LIN {X 0,Y 527.544,Z 904.757,A -85,B 0,C 180,E1 14975.921,E2 14975.921} C_VEL
LIN {X 0,Y 511.75,Z 974.005,A -85,B 0,C 180,E1 14979.243,E2 14979.243} C_VEL
LIN {X 0,Y 491.404,Z 1041.559,A -85,B 0,C 180,E1 14984.465,E2 14984.465} C_VEL
LIN {X 0,Y 471.066,Z 1101.33,A -85,B 0,C 180,E1 14991.676,E2 14991.676} C_VEL
LIN {X 0,Y 455.075,Z 1150.051,A -85,B 0,C 180,E1 15000.694,E2 15000.694} C_VEL
LIN {X 0,Y 446.451,Z 1183.071,A -85,B 0,C 180,E1 15010.14,E2 15010.14} C_VEL
LIN {X 0,Y 443.515,Z 1201.898,A -85,B 0,C 180,E1 15019.158,E2 15019.158} C_VEL
LIN {X 0,Y 443.252,Z 1209.224,A -85,B 0,C 180,E1 15027.056,E2 15027.056} C_VEL
LIN {X 0,Y 443.097,Z 1207.14,A -85,B 0,C 180,E1 15036.179,E2 15036.179} C_VEL
LIN {X 0,Y 443.595,Z 1202.243,A -85,B 0,C 180,E1 15040.591,E2 15040.591} C_VEL
LIN {X 0,Y 436.619,Z 1195.01,A -85,B 0,C 180,E1 15045.026,E2 15045.026} C_VEL
LIN {X 0,Y 442.886,Z 1167.282,A -85,B 0,C 180,E1 15055.338,E2 15055.338} C_VEL
LIN {X 0,Y 455.534,Z 1125.939,A -85,B 0,C 180,E1 15064.753,E2 15064.753} C_VEL
LIN {X 0,Y 473.85,Z 1072.374,A -85,B 0,C 180,E1 15072.653,E2 15072.653} C_VEL
LIN {X 0,Y 493.837,Z 1008.731,A -85,B 0,C 180,E1 15078.789,E2 15078.789} C_VEL
LIN {X 0,Y 512.572,Z 935.581,A -85,B 0,C 180,E1 15083.187,E2 15083.187} C_VEL
LIN {X 0,Y 518.028,Z 903.153,A -85,B 0,C 180,E1 15084.629,E2 15084.629} C_VEL
LIN {X 0,Y 493.673,Z 851.518,A -85,B 0,C 180,E1 15091.51,E2 15091.51} C_VEL
LIN {X 0,Y 466.915,Z 810.429,A -85,B 0,C 180,E1 15099.517,E2 15099.517} C_VEL
LIN {X 0,Y 448.656,Z 787.138,A -85,B 0,C 180,E1 15107.046,E2 15107.046} C_VEL
LIN {X 0,Y 439.151,Z 774.402,A -85,B 0,C 180,E1 15113.435,E2 15113.435} C_VEL
LIN {X 0,Y 434.536,Z 767.06,A -85,B 0,C 180,E1 15121.02,E2 15121.02} C_VEL
LIN {X 0,Y 434.845,Z 769.422,A -85,B 0,C 180,E1 15127.285,E2 15127.285} C_VEL
LIN {X 0,Y 441.325,Z 777.842,A -85,B 0,C 180,E1 15134.513,E2 15134.513} C_VEL
LIN {X 0,Y 452.767,Z 792.076,A -85,B 0,C 180,E1 15141.061,E2 15141.061} C_VEL
LIN {X 0,Y 474.863,Z 822.437,A -85,B 0,C 180,E1 15149.239,E2 15149.239} C_VEL
LIN {X 0,Y 501.419,Z 867.679,A -85,B 0,C 180,E1 15156.98,E2 15156.98} C_VEL
LIN {X 0,Y 517.133,Z 907.005,A -85,B 0,C 180,E1 15161.858,E2 15161.858} C_VEL
LIN {X 0,Y 499.871,Z 981.761,A -85,B 0,C 180,E1 15165.794,E2 15165.794} C_VEL
LIN {X 0,Y 479.961,Z 1047.78,A -85,B 0,C 180,E1 15171.441,E2 15171.441} C_VEL
LIN {X 0,Y 460.575,Z 1103.811,A -85,B 0,C 180,E1 15178.811,E2 15178.811} C_VEL
LIN {X 0,Y 446.089,Z 1147.116,A -85,B 0,C 180,E1 15187.518,E2 15187.518} C_VEL
LIN {X 0,Y 438.118,Z 1178.477,A -85,B 0,C 180,E1 15197.509,E2 15197.509} C_VEL
LIN {X 0,Y 435.402,Z 1195.059,A -85,B 0,C 180,E1 15207.008,E2 15207.008} C_VEL
LIN {X 0,Y 434.743,Z 1200.24,A -85,B 0,C 180,E1 15215.88,E2 15215.88} C_VEL
LIN {X 0,Y 435.395,Z 1194.776,A -85,B 0,C 180,E1 15225.145,E2 15225.145} C_VEL
LIN {X 0,Y 437.899,Z 1178.172,A -85,B 0,C 180,E1 15234.558,E2 15234.558} C_VEL
LIN {X 0,Y 446.288,Z 1146.664,A -85,B 0,C 180,E1 15244.563,E2 15244.563} C_VEL
LIN {X 0,Y 462.337,Z 1100.95,A -85,B 0,C 180,E1 15253.74,E2 15253.74} C_VEL
LIN {X 0,Y 483.029,Z 1043.534,A -85,B 0,C 180,E1 15261.229,E2 15261.229} C_VEL
LIN {X 0,Y 504.194,Z 977.942,A -85,B 0,C 180,E1 15266.717,E2 15266.717} C_VEL
LIN {X 0,Y 521.526,Z 904.091,A -85,B 0,C 180,E1 15270.64,E2 15270.64} C_VEL
LIN {X 0,Y 503.397,Z 862.252,A -85,B 0,C 180,E1 15277.068,E2 15277.068} C_VEL
LIN {X 0,Y 482.023,Z 826.723,A -85,B 0,C 180,E1 15285.517,E2 15285.517} C_VEL
LIN {X 0,Y 470.998,Z 812.054,A -85,B 0,C 180,E1 15291.649,E2 15291.649} C_VEL
LIN {X 0,Y 464.92,Z 803.945,A -85,B 0,C 180,E1 15297.527,E2 15297.527} C_VEL
LIN {X 0,Y 463.82,Z 803.136,A -85,B 0,C 180,E1 15306.379,E2 15306.379} C_VEL
LIN {X 0,Y 468.95,Z 809.648,A -85,B 0,C 180,E1 15312.592,E2 15312.592} C_VEL
LIN {X 0,Y 482.636,Z 828.099,A -85,B 0,C 180,E1 15320.554,E2 15320.554} C_VEL
LIN {X 0,Y 504.042,Z 862.875,A -85,B 0,C 180,E1 15328.764,E2 15328.764} C_VEL
LIN {X 0,Y 522.75,Z 905.365,A -85,B 0,C 180,E1 15335.174,E2 15335.174} C_VEL
LIN {X 0,Y 505.795,Z 977.464,A -85,B 0,C 180,E1 15338.719,E2 15338.719} C_VEL
LIN {X 0,Y 484.736,Z 1044.49,A -85,B 0,C 180,E1 15344.039,E2 15344.039} C_VEL
LIN {X 0,Y 463.733,Z 1103.615,A -85,B 0,C 180,E1 15351.37,E2 15351.37} C_VEL
LIN {X 0,Y 447.299,Z 1151.661,A -85,B 0,C 180,E1 15360.552,E2 15360.552} C_VEL
LIN {X 0,Y 438.391,Z 1184.327,A -85,B 0,C 180,E1 15370.287,E2 15370.287} C_VEL
LIN {X 0,Y 435.524,Z 1203.155,A -85,B 0,C 180,E1 15379.971,E2 15379.971} C_VEL
LIN {X 0,Y 434.854,Z 1209.594,A -85,B 0,C 180,E1 15388.998,E2 15388.998} C_VEL
LIN {X 0,Y 435.348,Z 1205.605,A -85,B 0,C 180,E1 15398.006,E2 15398.006} C_VEL
LIN {X 0,Y 436.619,Z 1195.01,A -85,B 0,C 180,E1 15405.026,E2 15405.026} C_VEL
LIN {X 0,Y 430.284,Z 1185.776,A -85,B 0,C 180,E1 15409.498,E2 15409.498} C_VEL
LIN {X 0,Y 438.823,Z 1154.658,A -85,B 0,C 180,E1 15419.214,E2 15419.214} C_VEL
LIN {X 0,Y 454.204,Z 1109.758,A -85,B 0,C 180,E1 15428.142,E2 15428.142} C_VEL
LIN {X 0,Y 474.682,Z 1051.658,A -85,B 0,C 180,E1 15435.636,E2 15435.636} C_VEL
LIN {X 0,Y 495.245,Z 985.357,A -85,B 0,C 180,E1 15441.128,E2 15441.128} C_VEL
LIN {X 0,Y 512.301,Z 911.314,A -85,B 0,C 180,E1 15444.954,E2 15444.954} C_VEL
LIN {X 0,Y 505.431,Z 889.358,A -85,B 0,C 180,E1 15447.387,E2 15447.387} C_VEL
LIN {X 0,Y 480.797,Z 841.969,A -85,B 0,C 180,E1 15454.624,E2 15454.624} C_VEL
LIN {X 0,Y 455.242,Z 804.445,A -85,B 0,C 180,E1 15463.505,E2 15463.505} C_VEL
LIN {X 0,Y 442.161,Z 788.381,A -85,B 0,C 180,E1 15470.268,E2 15470.268} C_VEL
LIN {X 0,Y 436.989,Z 781.618,A -85,B 0,C 180,E1 15474.48,E2 15474.48} C_VEL
LIN {X 0,Y 433.262,Z 774.957,A -85,B 0,C 180,E1 15481.023,E2 15481.023} C_VEL
LIN {X 0,Y 433.828,Z 777.457,A -85,B 0,C 180,E1 15487.239,E2 15487.239} C_VEL
LIN {X 0,Y 440.096,Z 785.808,A -85,B 0,C 180,E1 15494.363,E2 15494.363} C_VEL
LIN {X 0,Y 451.617,Z 800.627,A -85,B 0,C 180,E1 15501.043,E2 15501.043} C_VEL
LIN {X 0,Y 473.311,Z 830.704,A -85,B 0,C 180,E1 15509.212,E2 15509.212} C_VEL
LIN {X 0,Y 498.779,Z 876.898,A -85,B 0,C 180,E1 15517.073,E2 15517.073} C_VEL
LIN {X 0,Y 511.431,Z 910.667,A -85,B 0,C 180,E1 15521.291,E2 15521.291} C_VEL
LIN {X 0,Y 493.793,Z 984.11,A -85,B 0,C 180,E1 15525.246,E2 15525.246} C_VEL
LIN {X 0,Y 473.502,Z 1049.051,A -85,B 0,C 180,E1 15530.894,E2 15530.894} C_VEL
LIN {X 0,Y 453.223,Z 1105.566,A -85,B 0,C 180,E1 15538.483,E2 15538.483} C_VEL
LIN {X 0,Y 438.006,Z 1149.456,A -85,B 0,C 180,E1 15547.617,E2 15547.617} C_VEL
LIN {X 0,Y 430.082,Z 1179.925,A -85,B 0,C 180,E1 15557.789,E2 15557.789} C_VEL
LIN {X 0,Y 427.417,Z 1195.277,A -85,B 0,C 180,E1 15566.952,E2 15566.952} C_VEL
LIN {X 0,Y 426.81,Z 1200.196,A -85,B 0,C 180,E1 15575.099,E2 15575.099} C_VEL
LIN {X 0,Y 427.323,Z 1195.951,A -85,B 0,C 180,E1 15584.387,E2 15584.387} C_VEL
LIN {X 0,Y 429.624,Z 1180.354,A -85,B 0,C 180,E1 15593.952,E2 15593.952} C_VEL
LIN {X 0,Y 437.425,Z 1151.263,A -85,B 0,C 180,E1 15603.897,E2 15603.897} C_VEL
LIN {X 0,Y 453.268,Z 1107.536,A -85,B 0,C 180,E1 15613.306,E2 15613.306} C_VEL
LIN {X 0,Y 474.327,Z 1051.817,A -85,B 0,C 180,E1 15621.071,E2 15621.071} C_VEL
LIN {X 0,Y 496.382,Z 987.421,A -85,B 0,C 180,E1 15626.816,E2 15626.816} C_VEL
LIN {X 0,Y 515.365,Z 915.073,A -85,B 0,C 180,E1 15630.847,E2 15630.847} C_VEL
LIN {X 0,Y 515.415,Z 904.877,A -85,B 0,C 180,E1 15631.65,E2 15631.65} C_VEL
LIN {X 0,Y 497.403,Z 863.792,A -85,B 0,C 180,E1 15638.404,E2 15638.404} C_VEL
LIN {X 0,Y 478.243,Z 831.882,A -85,B 0,C 180,E1 15646.629,E2 15646.629} C_VEL
LIN {X 0,Y 469.042,Z 819.224,A -85,B 0,C 180,E1 15652.198,E2 15652.198} C_VEL
LIN {X 0,Y 463.68,Z 811.675,A -85,B 0,C 180,E1 15657.872,E2 15657.872} C_VEL
LIN {X 0,Y 462.866,Z 811.161,A -85,B 0,C 180,E1 15666.449,E2 15666.449} C_VEL
LIN {X 0,Y 467.768,Z 817.729,A -85,B 0,C 180,E1 15672.565,E2 15672.565} C_VEL
LIN {X 0,Y 480.999,Z 836.391,A -85,B 0,C 180,E1 15680.49,E2 15680.49} C_VEL
LIN {X 0,Y 500.903,Z 869.793,A -85,B 0,C 180,E1 15688.467,E2 15688.467} C_VEL
LIN {X 0,Y 517.594,Z 910.088,A -85,B 0,C 180,E1 15694.62,E2 15694.62} C_VEL
LIN {X 0,Y 500.186,Z 979.931,A -85,B 0,C 180,E1 15698.123,E2 15698.123} C_VEL
LIN {X 0,Y 478.85,Z 1045.335,A -85,B 0,C 180,E1 15703.392,E2 15703.392} C_VEL
LIN {X 0,Y 457.12,Z 1104.142,A -85,B 0,C 180,E1 15710.784,E2 15710.784} C_VEL
LIN {X 0,Y 439.997,Z 1151.661,A -85,B 0,C 180,E1 15720.014,E2 15720.014} C_VEL
LIN {X 0,Y 430.592,Z 1184.406,A -85,B 0,C 180,E1 15729.983,E2 15729.983} C_VEL
LIN {X 0,Y 427.55,Z 1203.064,A -85,B 0,C 180,E1 15739.782,E2 15739.782} C_VEL
LIN {X 0,Y 426.881,Z 1209.506,A -85,B 0,C 180,E1 15748.979,E2 15748.979} C_VEL
LIN {X 0,Y 427.369,Z 1205.518,A -85,B 0,C 180,E1 15758.157,E2 15758.157} C_VEL
LIN {X 0,Y 429.73,Z 1189.27,A -85,B 0,C 180,E1 15768.005,E2 15768.005} C_VEL
LIN {X 0,Y 430.284,Z 1185.776,A -85,B 0,C 180,E1 15769.498,E2 15769.498} C_VEL
LIN {X 0,Y 425.732,Z 1174.46,A -85,B 0,C 180,E1 15773.967,E2 15773.967} C_VEL
LIN {X 0,Y 438.451,Z 1135.512,A -85,B 0,C 180,E1 15784.015,E2 15784.015} C_VEL
LIN {X 0,Y 456.719,Z 1085.237,A -85,B 0,C 180,E1 15792.343,E2 15792.343} C_VEL
LIN {X 0,Y 477.879,Z 1024.143,A -85,B 0,C 180,E1 15798.932,E2 15798.932} C_VEL
LIN {X 0,Y 498.355,Z 953.286,A -85,B 0,C 180,E1 15803.739,E2 15803.739} C_VEL
LIN {X 0,Y 506.726,Z 909.72,A -85,B 0,C 180,E1 15805.888,E2 15805.888} C_VEL
LIN {X 0,Y 484.061,Z 859.821,A -85,B 0,C 180,E1 15812.996,E2 15812.996} C_VEL
LIN {X 0,Y 460.14,Z 821.877,A -85,B 0,C 180,E1 15821.022,E2 15821.022} C_VEL
LIN {X 0,Y 442.558,Z 797.464,A -85,B 0,C 180,E1 15829.404,E2 15829.404} C_VEL
LIN {X 0,Y 434.802,Z 788.415,A -85,B 0,C 180,E1 15835.769,E2 15835.769} C_VEL
LIN {X 0,Y 432.036,Z 782.793,A -85,B 0,C 180,E1 15843.039,E2 15843.039} C_VEL
LIN {X 0,Y 433.2,Z 786.627,A -85,B 0,C 180,E1 15848.072,E2 15848.072} C_VEL
LIN {X 0,Y 438.953,Z 793.854,A -85,B 0,C 180,E1 15854.274,E2 15854.274} C_VEL
LIN {X 0,Y 450.772,Z 809.434,A -85,B 0,C 180,E1 15861.159,E2 15861.159} C_VEL
LIN {X 0,Y 471.107,Z 838.906,A -85,B 0,C 180,E1 15869.098,E2 15869.098} C_VEL
LIN {X 0,Y 495.448,Z 884.581,A -85,B 0,C 180,E1 15876.952,E2 15876.952} C_VEL
LIN {X 0,Y 505.883,Z 913.865,A -85,B 0,C 180,E1 15880.694,E2 15880.694} C_VEL
LIN {X 0,Y 487.255,Z 988.086,A -85,B 0,C 180,E1 15884.798,E2 15884.798} C_VEL
LIN {X 0,Y 466.143,Z 1052.978,A -85,B 0,C 180,E1 15890.63,E2 15890.63} C_VEL
LIN {X 0,Y 445.362,Z 1108.798,A -85,B 0,C 180,E1 15898.403,E2 15898.403} C_VEL
LIN {X 0,Y 429.945,Z 1151.782,A -85,B 0,C 180,E1 15907.721,E2 15907.721} C_VEL
LIN {X 0,Y 422.01,Z 1181.37,A -85,B 0,C 180,E1 15918.079,E2 15918.079} C_VEL
LIN {X 0,Y 419.433,Z 1195.494,A -85,B 0,C 180,E1 15926.894,E2 15926.894} C_VEL
LIN {X 0,Y 418.8,Z 1200.302,A -85,B 0,C 180,E1 15935.197,E2 15935.197} C_VEL
LIN {X 0,Y 419.367,Z 1195.906,A -85,B 0,C 180,E1 15944.666,E2 15944.666} C_VEL
LIN {X 0,Y 421.862,Z 1180.194,A -85,B 0,C 180,E1 15954.421,E2 15954.421} C_VEL
LIN {X 0,Y 430.332,Z 1150.826,A -85,B 0,C 180,E1 15964.584,E2 15964.584} C_VEL
LIN {X 0,Y 447.524,Z 1105.761,A -85,B 0,C 180,E1 15974.313,E2 15974.313} C_VEL
LIN {X 0,Y 469.644,Z 1049.427,A -85,B 0,C 180,E1 15982.099,E2 15982.099} C_VEL
LIN {X 0,Y 492.139,Z 985.474,A -85,B 0,C 180,E1 15987.725,E2 15987.725} C_VEL
LIN {X 0,Y 511.167,Z 914.54,A -85,B 0,C 180,E1 15991.634,E2 15991.634} C_VEL
LIN {X 0,Y 498.544,Z 879.538,A -85,B 0,C 180,E1 15996.978,E2 15996.978} C_VEL
LIN {X 0,Y 480.407,Z 846.259,A -85,B 0,C 180,E1 16004.706,E2 16004.706} C_VEL
LIN {X 0,Y 468.686,Z 828.027,A -85,B 0,C 180,E1 16011.607,E2 16011.607} C_VEL
LIN {X 0,Y 462.377,Z 819.472,A -85,B 0,C 180,E1 16018.101,E2 16018.101} C_VEL
LIN {X 0,Y 461.67,Z 819.022,A -85,B 0,C 180,E1 16026.348,E2 16026.348} C_VEL
LIN {X 0,Y 466.535,Z 825.804,A -85,B 0,C 180,E1 16032.539,E2 16032.539} C_VEL
LIN {X 0,Y 479.328,Z 844.724,A -85,B 0,C 180,E1 16040.496,E2 16040.496} C_VEL
LIN {X 0,Y 497.797,Z 877.026,A -85,B 0,C 180,E1 16048.241,E2 16048.241} C_VEL
LIN {X 0,Y 512.578,Z 913.238,A -85,B 0,C 180,E1 16053.968,E2 16053.968} C_VEL
LIN {X 0,Y 493.972,Z 984.794,A -85,B 0,C 180,E1 16057.669,E2 16057.669} C_VEL
LIN {X 0,Y 471.585,Z 1050.203,A -85,B 0,C 180,E1 16063.136,E2 16063.136} C_VEL
LIN {X 0,Y 448.925,Z 1108.735,A -85,B 0,C 180,E1 16070.808,E2 16070.808} C_VEL
LIN {X 0,Y 431.71,Z 1154.894,A -85,B 0,C 180,E1 16080.25,E2 16080.25} C_VEL
LIN {X 0,Y 422.531,Z 1185.514,A -85,B 0,C 180,E1 16090.062,E2 16090.062} C_VEL
LIN {X 0,Y 419.569,Z 1202.973,A -85,B 0,C 180,E1 16099.586,E2 16099.586} C_VEL
LIN {X 0,Y 418.883,Z 1209.419,A -85,B 0,C 180,E1 16108.96,E2 16108.96} C_VEL
LIN {X 0,Y 419.408,Z 1205.43,A -85,B 0,C 180,E1 16118.313,E2 16118.313} C_VEL
LIN {X 0,Y 422.039,Z 1188.061,A -85,B 0,C 180,E1 16128.865,E2 16128.865} C_VEL
LIN {X 0,Y 425.732,Z 1174.46,A -85,B 0,C 180,E1 16133.967,E2 16133.967} C_VEL
LIN {X 0,Y 421.79,Z 1161.371,A -85,B 0,C 180,E1 16138.405,E2 16138.405} C_VEL
LIN {X 0,Y 437.412,Z 1118.507,A -85,B 0,C 180,E1 16147.892,E2 16147.892} C_VEL
LIN {X 0,Y 458.873,Z 1062.37,A -85,B 0,C 180,E1 16155.849,E2 16155.849} C_VEL
LIN {X 0,Y 480.999,Z 997.028,A -85,B 0,C 180,E1 16161.776,E2 16161.776} C_VEL
LIN {X 0,Y 500.266,Z 922.469,A -85,B 0,C 180,E1 16165.96,E2 16165.96} C_VEL
LIN {X 0,Y 500.637,Z 911.67,A -85,B 0,C 180,E1 16166.71,E2 16166.71} C_VEL
LIN {X 0,Y 478.937,Z 863.359,A -85,B 0,C 180,E1 16173.88,E2 16173.88} C_VEL
LIN {X 0,Y 455.425,Z 825.158,A -85,B 0,C 180,E1 16182.389,E2 16182.389} C_VEL
LIN {X 0,Y 439.883,Z 804.177,A -85,B 0,C 180,E1 16190.436,E2 16190.436} C_VEL
LIN {X 0,Y 433.62,Z 796.145,A -85,B 0,C 180,E1 16196.008,E2 16196.008} C_VEL
LIN {X 0,Y 431.06,Z 790.732,A -85,B 0,C 180,E1 16203.046,E2 16203.046} C_VEL
LIN {X 0,Y 432.823,Z 795.687,A -85,B 0,C 180,E1 16209.094,E2 16209.094} C_VEL
LIN {X 0,Y 437.834,Z 801.912,A -85,B 0,C 180,E1 16214.201,E2 16214.201} C_VEL
LIN {X 0,Y 451.778,Z 820.251,A -85,B 0,C 180,E1 16222.181,E2 16222.181} C_VEL
LIN {X 0,Y 474.385,Z 856.439,A -85,B 0,C 180,E1 16230.916,E2 16230.916} C_VEL
LIN {X 0,Y 497.356,Z 905.62,A -85,B 0,C 180,E1 16238.721,E2 16238.721} C_VEL
LIN {X 0,Y 500.226,Z 917.865,A -85,B 0,C 180,E1 16240.12,E2 16240.12} C_VEL
LIN {X 0,Y 480.931,Z 991.452,A -85,B 0,C 180,E1 16244.296,E2 16244.296} C_VEL
LIN {X 0,Y 459.148,Z 1055.933,A -85,B 0,C 180,E1 16250.249,E2 16250.249} C_VEL
LIN {X 0,Y 437.986,Z 1110.694,A -85,B 0,C 180,E1 16258.086,E2 16258.086} C_VEL
LIN {X 0,Y 421.892,Z 1154.099,A -85,B 0,C 180,E1 16267.83,E2 16267.83} C_VEL
LIN {X 0,Y 413.875,Z 1182.805,A -85,B 0,C 180,E1 16278.377,E2 16278.377} C_VEL
LIN {X 0,Y 411.465,Z 1195.711,A -85,B 0,C 180,E1 16286.834,E2 16286.834} C_VEL
LIN {X 0,Y 410.785,Z 1200.408,A -85,B 0,C 180,E1 16295.298,E2 16295.298} C_VEL
LIN {X 0,Y 411.379,Z 1195.859,A -85,B 0,C 180,E1 16304.957,E2 16304.957} C_VEL
LIN {X 0,Y 414.143,Z 1180.054,A -85,B 0,C 180,E1 16314.907,E2 16314.907} C_VEL
LIN {X 0,Y 423.337,Z 1150.332,A -85,B 0,C 180,E1 16325.315,E2 16325.315} C_VEL
LIN {X 0,Y 440.76,Z 1106.751,A -85,B 0,C 180,E1 16334.859,E2 16334.859} C_VEL
LIN {X 0,Y 463.632,Z 1050.744,A -85,B 0,C 180,E1 16342.729,E2 16342.729} C_VEL
LIN {X 0,Y 487.113,Z 986.243,A -85,B 0,C 180,E1 16348.46,E2 16348.46} C_VEL
LIN {X 0,Y 505.811,Z 914.579,A -85,B 0,C 180,E1 16352.623,E2 16352.623} C_VEL
LIN {X 0,Y 489.942,Z 875.591,A -85,B 0,C 180,E1 16359.42,E2 16359.42} C_VEL
LIN {X 0,Y 472.195,Z 842.896,A -85,B 0,C 180,E1 16368.282,E2 16368.282} C_VEL
LIN {X 0,Y 461.973,Z 828.408,A -85,B 0,C 180,E1 16376.927,E2 16376.927} C_VEL
LIN {X 0,Y 460.317,Z 826.496,A -85,B 0,C 180,E1 16385.773,E2 16385.773} C_VEL
LIN {X 0,Y 465.1,Z 833.568,A -85,B 0,C 180,E1 16392.398,E2 16392.398} C_VEL
LIN {X 0,Y 477.435,Z 852.633,A -85,B 0,C 180,E1 16400.393,E2 16400.393} C_VEL
LIN {X 0,Y 494.594,Z 884.402,A -85,B 0,C 180,E1 16408.041,E2 16408.041} C_VEL
LIN {X 0,Y 507.132,Z 918.331,A -85,B 0,C 180,E1 16413.4,E2 16413.4} C_VEL
LIN {X 0,Y 487.778,Z 989.155,A -85,B 0,C 180,E1 16417.184,E2 16417.184} C_VEL
LIN {X 0,Y 464.681,Z 1053.822,A -85,B 0,C 180,E1 16422.75,E2 16422.75} C_VEL
LIN {X 0,Y 441.213,Z 1111.854,A -85,B 0,C 180,E1 16430.641,E2 16430.641} C_VEL
LIN {X 0,Y 424.097,Z 1155.884,A -85,B 0,C 180,E1 16439.957,E2 16439.957} C_VEL
LIN {X 0,Y 414.453,Z 1186.807,A -85,B 0,C 180,E1 16450.214,E2 16450.214} C_VEL
LIN {X 0,Y 411.523,Z 1204.11,A -85,B 0,C 180,E1 16460.452,E2 16460.452} C_VEL
LIN {X 0,Y 410.892,Z 1209.331,A -85,B 0,C 180,E1 16468.94,E2 16468.94} C_VEL
LIN {X 0,Y 411.451,Z 1205.343,A -85,B 0,C 180,E1 16478.475,E2 16478.475} C_VEL
LIN {X 0,Y 413.989,Z 1189.107,A -85,B 0,C 180,E1 16488.691,E2 16488.691} C_VEL
LIN {X 0,Y 421.79,Z 1161.371,A -85,B 0,C 180,E1 16498.405,E2 16498.405} C_VEL
LIN {X 0,Y 420.153,Z 1146.311,A -85,B 0,C 180,E1 16502.778,E2 16502.778} C_VEL
LIN {X 0,Y 439.363,Z 1097.233,A -85,B 0,C 180,E1 16512.009,E2 16512.009} C_VEL
LIN {X 0,Y 462.223,Z 1037.268,A -85,B 0,C 180,E1 16519.197,E2 16519.197} C_VEL
LIN {X 0,Y 484.261,Z 968.826,A -85,B 0,C 180,E1 16524.354,E2 16524.354} C_VEL
LIN {X 0,Y 495.901,Z 917.508,A -85,B 0,C 180,E1 16527.03,E2 16527.03} C_VEL
LIN {X 0,Y 475.617,Z 870.172,A -85,B 0,C 180,E1 16534.201,E2 16534.201} C_VEL
LIN {X 0,Y 453.367,Z 832.508,A -85,B 0,C 180,E1 16542.699,E2 16542.699} C_VEL
LIN {X 0,Y 438.359,Z 811.746,A -85,B 0,C 180,E1 16550.78,E2 16550.78} C_VEL
LIN {X 0,Y 431.822,Z 802.803,A -85,B 0,C 180,E1 16557.165,E2 16557.165} C_VEL
LIN {X 0,Y 430.083,Z 798.671,A -85,B 0,C 180,E1 16563.053,E2 16563.053} C_VEL
LIN {X 0,Y 435.48,Z 807.032,A -85,B 0,C 180,E1 16572.978,E2 16572.978} C_VEL
LIN {X 0,Y 450.962,Z 829.824,A -85,B 0,C 180,E1 16582.436,E2 16582.436} C_VEL
LIN {X 0,Y 471.185,Z 863.38,A -85,B 0,C 180,E1 16590.603,E2 16590.603} C_VEL
LIN {X 0,Y 492.677,Z 911.482,A -85,B 0,C 180,E1 16598.395,E2 16598.395} C_VEL
LIN {X 0,Y 494.395,Z 923.157,A -85,B 0,C 180,E1 16599.596,E2 16599.596} C_VEL
LIN {X 0,Y 473.914,Z 997.167,A -85,B 0,C 180,E1 16603.952,E2 16603.952} C_VEL
LIN {X 0,Y 451.51,Z 1060.51,A -85,B 0,C 180,E1 16610.037,E2 16610.037} C_VEL
LIN {X 0,Y 429.957,Z 1114.331,A -85,B 0,C 180,E1 16618.076,E2 16618.076} C_VEL
LIN {X 0,Y 413.797,Z 1156.337,A -85,B 0,C 180,E1 16627.94,E2 16627.94} C_VEL
LIN {X 0,Y 405.727,Z 1184.225,A -85,B 0,C 180,E1 16638.687,E2 16638.687} C_VEL
LIN {X 0,Y 403.005,Z 1197.79,A -85,B 0,C 180,E1 16648.925,E2 16648.925} C_VEL
LIN {X 0,Y 402.719,Z 1200.348,A -85,B 0,C 180,E1 16657.576,E2 16657.576} C_VEL
LIN {X 0,Y 403.724,Z 1193.376,A -85,B 0,C 180,E1 16667.489,E2 16667.489} C_VEL
LIN {X 0,Y 408.956,Z 1172.582,A -85,B 0,C 180,E1 16678.557,E2 16678.557} C_VEL
LIN {X 0,Y 421.761,Z 1137.242,A -85,B 0,C 180,E1 16689.321,E2 16689.321} C_VEL
LIN {X 0,Y 442.298,Z 1088.892,A -85,B 0,C 180,E1 16698.546,E2 16698.546} C_VEL
LIN {X 0,Y 466.66,Z 1029.501,A -85,B 0,C 180,E1 16705.754,E2 16705.754} C_VEL
LIN {X 0,Y 490.559,Z 960.873,A -85,B 0,C 180,E1 16710.902,E2 16710.902} C_VEL
LIN {X 0,Y 500.922,Z 918.973,A -85,B 0,C 180,E1 16713.186,E2 16713.186} C_VEL
LIN {X 0,Y 485.66,Z 880.251,A -85,B 0,C 180,E1 16720.184,E2 16720.184} C_VEL
LIN {X 0,Y 469.477,Z 849.676,A -85,B 0,C 180,E1 16728.921,E2 16728.921} C_VEL
LIN {X 0,Y 460.316,Z 835.967,A -85,B 0,C 180,E1 16737.266,E2 16737.266} C_VEL
LIN {X 0,Y 459.04,Z 834.525,A -85,B 0,C 180,E1 16745.908,E2 16745.908} C_VEL
LIN {X 0,Y 463.635,Z 841.779,A -85,B 0,C 180,E1 16752.498,E2 16752.498} C_VEL
LIN {X 0,Y 475.21,Z 860.414,A -85,B 0,C 180,E1 16760.292,E2 16760.292} C_VEL
LIN {X 0,Y 491.589,Z 892.022,A -85,B 0,C 180,E1 16767.904,E2 16767.904} C_VEL
LIN {X 0,Y 501.805,Z 922.975,A -85,B 0,C 180,E1 16772.792,E2 16772.792} C_VEL
LIN {X 0,Y 481.27,Z 994.362,A -85,B 0,C 180,E1 16776.749,E2 16776.749} C_VEL
LIN {X 0,Y 457.389,Z 1058.243,A -85,B 0,C 180,E1 16782.464,E2 16782.464} C_VEL
LIN {X 0,Y 433.288,Z 1115.467,A -85,B 0,C 180,E1 16790.564,E2 16790.564} C_VEL
LIN {X 0,Y 415.39,Z 1159.804,A -85,B 0,C 180,E1 16800.469,E2 16800.469} C_VEL
LIN {X 0,Y 406.1,Z 1189.088,A -85,B 0,C 180,E1 16810.926,E2 16810.926} C_VEL
LIN {X 0,Y 403.508,Z 1205.24,A -85,B 0,C 180,E1 16821.351,E2 16821.351} C_VEL
LIN {X 0,Y 402.894,Z 1209.244,A -85,B 0,C 180,E1 16828.919,E2 16828.919} C_VEL
LIN {X 0,Y 403.488,Z 1205.25,A -85,B 0,C 180,E1 16838.643,E2 16838.643} C_VEL
LIN {X 0,Y 406.143,Z 1188.976,A -85,B 0,C 180,E1 16849.066,E2 16849.066} C_VEL
LIN {X 0,Y 415.172,Z 1159.048,A -85,B 0,C 180,E1 16859.541,E2 16859.541} C_VEL
LIN {X 0,Y 420.153,Z 1146.311,A -85,B 0,C 180,E1 16862.778,E2 16862.778} C_VEL
LIN {X 0,Y 419.459,Z 1129.544,A -85,B 0,C 180,E1 16867.061,E2 16867.061} C_VEL
LIN {X 0,Y 441.429,Z 1076.454,A -85,B 0,C 180,E1 16875.584,E2 16875.584} C_VEL
LIN {X 0,Y 464.863,Z 1013.543,A -85,B 0,C 180,E1 16882.041,E2 16882.041} C_VEL
LIN {X 0,Y 486.632,Z 940.619,A -85,B 0,C 180,E1 16886.638,E2 16886.638} C_VEL
LIN {X 0,Y 490.134,Z 920.388,A -85,B 0,C 180,E1 16887.756,E2 16887.756} C_VEL
LIN {X 0,Y 470.609,Z 873.605,A -85,B 0,C 180,E1 16895.121,E2 16895.121} C_VEL
LIN {X 0,Y 449.587,Z 837.691,A -85,B 0,C 180,E1 16903.67,E2 16903.67} C_VEL
LIN {X 0,Y 435.858,Z 818.143,A -85,B 0,C 180,E1 16911.766,E2 16911.766} C_VEL
LIN {X 0,Y 429.351,Z 806.717,A -85,B 0,C 180,E1 16921.032,E2 16921.032} C_VEL
LIN {X 0,Y 429.72,Z 809.189,A -85,B 0,C 180,E1 16926.862,E2 16926.862} C_VEL
LIN {X 0,Y 435.491,Z 817.992,A -85,B 0,C 180,E1 16934.103,E2 16934.103} C_VEL
LIN {X 0,Y 448.926,Z 837.488,A -85,B 0,C 180,E1 16942.26,E2 16942.26} C_VEL
LIN {X 0,Y 468.247,Z 870.977,A -85,B 0,C 180,E1 16950.423,E2 16950.423} C_VEL
LIN {X 0,Y 488.472,Z 918.723,A -85,B 0,C 180,E1 16958.26,E2 16958.26} C_VEL
LIN {X 0,Y 488.584,Z 927.95,A -85,B 0,C 180,E1 16959.048,E2 16959.048} C_VEL
LIN {X 0,Y 467.48,Z 1000.73,A -85,B 0,C 180,E1 16963.467,E2 16963.467} C_VEL
LIN {X 0,Y 444.588,Z 1063.032,A -85,B 0,C 180,E1 16969.607,E2 16969.607} C_VEL
LIN {X 0,Y 422.071,Z 1117.181,A -85,B 0,C 180,E1 16977.963,E2 16977.963} C_VEL
LIN {X 0,Y 405.687,Z 1158.4,A -85,B 0,C 180,E1 16988.053,E2 16988.053} C_VEL
LIN {X 0,Y 397.548,Z 1185.44,A -85,B 0,C 180,E1 16999.008,E2 16999.008} C_VEL
LIN {X 0,Y 395.009,Z 1197.96,A -85,B 0,C 180,E1 17008.903,E2 17008.903} C_VEL
LIN {X 0,Y 394.705,Z 1200.419,A -85,B 0,C 180,E1 17017.731,E2 17017.731} C_VEL
LIN {X 0,Y 395.817,Z 1193.328,A -85,B 0,C 180,E1 17027.852,E2 17027.852} C_VEL
LIN {X 0,Y 401.364,Z 1172.581,A -85,B 0,C 180,E1 17039.083,E2 17039.083} C_VEL
LIN {X 0,Y 414.995,Z 1136.976,A -85,B 0,C 180,E1 17050.091,E2 17050.091} C_VEL
LIN {X 0,Y 436.769,Z 1088.085,A -85,B 0,C 180,E1 17059.453,E2 17059.453} C_VEL
LIN {X 0,Y 461.873,Z 1028.841,A -85,B 0,C 180,E1 17066.636,E2 17066.636} C_VEL
LIN {X 0,Y 486.427,Z 960.05,A -85,B 0,C 180,E1 17071.768,E2 17071.768} C_VEL
LIN {X 0,Y 495.785,Z 922.606,A -85,B 0,C 180,E1 17073.889,E2 17073.889} C_VEL
LIN {X 0,Y 481.327,Z 884.77,A -85,B 0,C 180,E1 17081.016,E2 17081.016} C_VEL
LIN {X 0,Y 466.483,Z 856.148,A -85,B 0,C 180,E1 17089.62,E2 17089.62} C_VEL
LIN {X 0,Y 458.581,Z 843.551,A -85,B 0,C 180,E1 17097.611,E2 17097.611} C_VEL
LIN {X 0,Y 457.561,Z 842.511,A -85,B 0,C 180,E1 17106.047,E2 17106.047} C_VEL
LIN {X 0,Y 462.189,Z 849.889,A -85,B 0,C 180,E1 17112.597,E2 17112.597} C_VEL
LIN {X 0,Y 474.108,Z 869.885,A -85,B 0,C 180,E1 17120.77,E2 17120.77} C_VEL
LIN {X 0,Y 490.168,Z 904.083,A -85,B 0,C 180,E1 17128.643,E2 17128.643} C_VEL
LIN {X 0,Y 496.8,Z 926.702,A -85,B 0,C 180,E1 17132.142,E2 17132.142} C_VEL
LIN {X 0,Y 475.193,Z 998.526,A -85,B 0,C 180,E1 17136.236,E2 17136.236} C_VEL
LIN {X 0,Y 450.205,Z 1062.444,A -85,B 0,C 180,E1 17142.143,E2 17142.143} C_VEL
LIN {X 0,Y 425.769,Z 1118.089,A -85,B 0,C 180,E1 17150.299,E2 17150.299} C_VEL
LIN {X 0,Y 407.605,Z 1161.209,A -85,B 0,C 180,E1 17160.281,E2 17160.281} C_VEL
LIN {X 0,Y 398.046,Z 1190.204,A -85,B 0,C 180,E1 17171.102,E2 17171.102} C_VEL
LIN {X 0,Y 395.523,Z 1205.165,A -85,B 0,C 180,E1 17181.175,E2 17181.175} C_VEL
LIN {X 0,Y 394.911,Z 1209.158,A -85,B 0,C 180,E1 17188.897,E2 17188.897} C_VEL
LIN {X 0,Y 395.511,Z 1205.149,A -85,B 0,C 180,E1 17198.819,E2 17198.819} C_VEL
LIN {X 0,Y 398.313,Z 1188.833,A -85,B 0,C 180,E1 17209.456,E2 17209.456} C_VEL
LIN {X 0,Y 407.876,Z 1158.836,A -85,B 0,C 180,E1 17220.124,E2 17220.124} C_VEL
LIN {X 0,Y 419.459,Z 1129.544,A -85,B 0,C 180,E1 17227.061,E2 17227.061} C_VEL
LIN {X 0,Y 420.6,Z 1111.036,A -85,B 0,C 180,E1 17231.191,E2 17231.191} C_VEL
LIN {X 0,Y 444.945,Z 1052.94,A -85,B 0,C 180,E1 17239.124,E2 17239.124} C_VEL
LIN {X 0,Y 468.774,Z 986.877,A -85,B 0,C 180,E1 17244.769,E2 17244.769} C_VEL
LIN {X 0,Y 484.795,Z 924.298,A -85,B 0,C 180,E1 17248.353,E2 17248.353} C_VEL
LIN {X 0,Y 466.369,Z 878.982,A -85,B 0,C 180,E1 17255.712,E2 17255.712} C_VEL
LIN {X 0,Y 446.609,Z 843.844,A -85,B 0,C 180,E1 17264.317,E2 17264.317} C_VEL
LIN {X 0,Y 432.631,Z 821.856,A -85,B 0,C 180,E1 17273.73,E2 17273.73} C_VEL
LIN {X 0,Y 428.051,Z 814.54,A -85,B 0,C 180,E1 17283.067,E2 17283.067} C_VEL
LIN {X 0,Y 433.156,Z 823.939,A -85,B 0,C 180,E1 17293.06,E2 17293.06} C_VEL
LIN {X 0,Y 446.523,Z 844.588,A -85,B 0,C 180,E1 17301.898,E2 17301.898} C_VEL
LIN {X 0,Y 464.733,Z 877.624,A -85,B 0,C 180,E1 17310.088,E2 17310.088} C_VEL
LIN {X 0,Y 483.965,Z 925.107,A -85,B 0,C 180,E1 17318.001,E2 17318.001} C_VEL
LIN {X 0,Y 463.01,Z 998.865,A -85,B 0,C 180,E1 17322.534,E2 17322.534} C_VEL
LIN {X 0,Y 439.296,Z 1061.792,A -85,B 0,C 180,E1 17328.689,E2 17328.689} C_VEL
LIN {X 0,Y 415.893,Z 1116.031,A -85,B 0,C 180,E1 17337.035,E2 17337.035} C_VEL
LIN {X 0,Y 398.758,Z 1157.075,A -85,B 0,C 180,E1 17347.061,E2 17347.061} C_VEL
LIN {X 0,Y 389.981,Z 1184.748,A -85,B 0,C 180,E1 17358.224,E2 17358.224} C_VEL
LIN {X 0,Y 387.024,Z 1198.125,A -85,B 0,C 180,E1 17368.881,E2 17368.881} C_VEL
LIN {X 0,Y 386.692,Z 1200.492,A -85,B 0,C 180,E1 17377.892,E2 17377.892} C_VEL
LIN {X 0,Y 387.907,Z 1193.277,A -85,B 0,C 180,E1 17388.228,E2 17388.228} C_VEL
LIN {X 0,Y 393.967,Z 1171.912,A -85,B 0,C 180,E1 17399.924,E2 17399.924} C_VEL
LIN {X 0,Y 408.706,Z 1135.772,A -85,B 0,C 180,E1 17411.104,E2 17411.104} C_VEL
LIN {X 0,Y 431.452,Z 1086.995,A -85,B 0,C 180,E1 17420.426,E2 17420.426} C_VEL
LIN {X 0,Y 456.961,Z 1028.829,A -85,B 0,C 180,E1 17427.477,E2 17427.477} C_VEL
LIN {X 0,Y 482.09,Z 960.387,A -85,B 0,C 180,E1 17432.58,E2 17432.58} C_VEL
LIN {X 0,Y 491.039,Z 927.511,A -85,B 0,C 180,E1 17434.398,E2 17434.398} C_VEL
LIN {X 0,Y 477.466,Z 890.4,A -85,B 0,C 180,E1 17441.609,E2 17441.609} C_VEL
LIN {X 0,Y 463.587,Z 862.495,A -85,B 0,C 180,E1 17450.327,E2 17450.327} C_VEL
LIN {X 0,Y 456.772,Z 851.029,A -85,B 0,C 180,E1 17458.078,E2 17458.078} C_VEL
LIN {X 0,Y 456.08,Z 850.603,A -85,B 0,C 180,E1 17466.221,E2 17466.221} C_VEL
LIN {X 0,Y 460.221,Z 857.605,A -85,B 0,C 180,E1 17472.472,E2 17472.472} C_VEL
LIN {X 0,Y 471.478,Z 877.274,A -85,B 0,C 180,E1 17480.583,E2 17480.583} C_VEL
LIN {X 0,Y 486.404,Z 910.655,A -85,B 0,C 180,E1 17488.336,E2 17488.336} C_VEL
LIN {X 0,Y 492.025,Z 929.71,A -85,B 0,C 180,E1 17491.444,E2 17491.444} C_VEL
LIN {X 0,Y 469.427,Z 1001.847,A -85,B 0,C 180,E1 17495.644,E2 17495.644} C_VEL
LIN {X 0,Y 443.535,Z 1065.502,A -85,B 0,C 180,E1 17501.68,E2 17501.68} C_VEL
LIN {X 0,Y 417.903,Z 1121.458,A -85,B 0,C 180,E1 17510.164,E2 17510.164} C_VEL
LIN {X 0,Y 398.969,Z 1164.661,A -85,B 0,C 180,E1 17520.716,E2 17520.716} C_VEL
LIN {X 0,Y 389.886,Z 1192.045,A -85,B 0,C 180,E1 17531.646,E2 17531.646} C_VEL
LIN {X 0,Y 387.365,Z 1205.967,A -85,B 0,C 180,E1 17542.121,E2 17542.121} C_VEL
LIN {X 0,Y 386.844,Z 1209.066,A -85,B 0,C 180,E1 17551.12,E2 17551.12} C_VEL
LIN {X 0,Y 387.698,Z 1202.598,A -85,B 0,C 180,E1 17561.267,E2 17561.267} C_VEL
LIN {X 0,Y 391.961,Z 1183.724,A -85,B 0,C 180,E1 17572.092,E2 17572.092} C_VEL
LIN {X 0,Y 404.173,Z 1150.267,A -85,B 0,C 180,E1 17582.955,E2 17582.955} C_VEL
LIN {X 0,Y 420.6,Z 1111.036,A -85,B 0,C 180,E1 17591.191,E2 17591.191} C_VEL
LIN {X 0,Y 423.338,Z 1090.632,A -85,B 0,C 180,E1 17595.125,E2 17595.125} C_VEL
LIN {X 0,Y 448.456,Z 1029.565,A -85,B 0,C 180,E1 17602.22,E2 17602.22} C_VEL
LIN {X 0,Y 472.209,Z 959.466,A -85,B 0,C 180,E1 17607.223,E2 17607.223} C_VEL
LIN {X 0,Y 479.772,Z 929.083,A -85,B 0,C 180,E1 17608.842,E2 17608.842} C_VEL
LIN {X 0,Y 462.46,Z 884.894,A -85,B 0,C 180,E1 17616.202,E2 17616.202} C_VEL
LIN {X 0,Y 443.501,Z 849.443,A -85,B 0,C 180,E1 17625.094,E2 17625.094} C_VEL
LIN {X 0,Y 430.935,Z 829.44,A -85,B 0,C 180,E1 17634.212,E2 17634.212} C_VEL
LIN {X 0,Y 426.895,Z 822.455,A -85,B 0,C 180,E1 17643.076,E2 17643.076} C_VEL
LIN {X 0,Y 432.024,Z 832.55,A -85,B 0,C 180,E1 17653.259,E2 17653.259} C_VEL
LIN {X 0,Y 444.609,Z 852.745,A -85,B 0,C 180,E1 17661.865,E2 17661.865} C_VEL
LIN {X 0,Y 461.909,Z 885.696,A -85,B 0,C 180,E1 17670.033,E2 17670.033} C_VEL
LIN {X 0,Y 478.605,Z 929.19,A -85,B 0,C 180,E1 17677.432,E2 17677.432} C_VEL
LIN {X 0,Y 457.134,Z 1001.061,A -85,B 0,C 180,E1 17681.903,E2 17681.903} C_VEL
LIN {X 0,Y 432.424,Z 1064.294,A -85,B 0,C 180,E1 17688.221,E2 17688.221} C_VEL
LIN {X 0,Y 408.407,Z 1118.022,A -85,B 0,C 180,E1 17696.724,E2 17696.724} C_VEL
LIN {X 0,Y 390.62,Z 1159.127,A -85,B 0,C 180,E1 17707.16,E2 17707.16} C_VEL
LIN {X 0,Y 381.778,Z 1185.939,A -85,B 0,C 180,E1 17718.548,E2 17718.548} C_VEL
LIN {X 0,Y 379.028,Z 1198.286,A -85,B 0,C 180,E1 17728.857,E2 17728.857} C_VEL
LIN {X 0,Y 378.679,Z 1200.565,A -85,B 0,C 180,E1 17738.06,E2 17738.06} C_VEL
LIN {X 0,Y 380.032,Z 1193.231,A -85,B 0,C 180,E1 17748.62,E2 17748.62} C_VEL
LIN {X 0,Y 386.466,Z 1171.753,A -85,B 0,C 180,E1 17760.567,E2 17760.567} C_VEL
LIN {X 0,Y 401.911,Z 1136.067,A -85,B 0,C 180,E1 17771.784,E2 17771.784} C_VEL
LIN {X 0,Y 425.844,Z 1086.813,A -85,B 0,C 180,E1 17781.291,E2 17781.291} C_VEL
LIN {X 0,Y 452.541,Z 1027.922,A -85,B 0,C 180,E1 17788.413,E2 17788.413} C_VEL
LIN {X 0,Y 478.104,Z 959.916,A -85,B 0,C 180,E1 17793.452,E2 17793.452} C_VEL
LIN {X 0,Y 485.979,Z 931.472,A -85,B 0,C 180,E1 17795.059,E2 17795.059} C_VEL
LIN {X 0,Y 473.441,Z 895.717,A -85,B 0,C 180,E1 17802.26,E2 17802.26} C_VEL
LIN {X 0,Y 460.561,Z 868.062,A -85,B 0,C 180,E1 17811.279,E2 17811.279} C_VEL
LIN {X 0,Y 454.466,Z 858.256,A -85,B 0,C 180,E1 17819.025,E2 17819.025} C_VEL
LIN {X 0,Y 454.383,Z 858.763,A -85,B 0,C 180,E1 17826.69,E2 17826.69} C_VEL
LIN {X 0,Y 459.424,Z 866.799,A -85,B 0,C 180,E1 17833.464,E2 17833.464} C_VEL
LIN {X 0,Y 471.966,Z 891.478,A -85,B 0,C 180,E1 17842.285,E2 17842.285} C_VEL
LIN {X 0,Y 485.182,Z 925.576,A -85,B 0,C 180,E1 17849.559,E2 17849.559} C_VEL
LIN {X 0,Y 486.507,Z 935.276,A -85,B 0,C 180,E1 17850.858,E2 17850.858} C_VEL
LIN {X 0,Y 462.854,Z 1007.027,A -85,B 0,C 180,E1 17855.192,E2 17855.192} C_VEL
LIN {X 0,Y 436.439,Z 1069.313,A -85,B 0,C 180,E1 17861.31,E2 17861.31} C_VEL
LIN {X 0,Y 410.702,Z 1123.181,A -85,B 0,C 180,E1 17869.743,E2 17869.743} C_VEL
LIN {X 0,Y 391.343,Z 1165.511,A -85,B 0,C 180,E1 17880.39,E2 17880.39} C_VEL
LIN {X 0,Y 382.057,Z 1191.865,A -85,B 0,C 180,E1 17891.175,E2 17891.175} C_VEL
LIN {X 0,Y 379.378,Z 1205.898,A -85,B 0,C 180,E1 17901.954,E2 17901.954} C_VEL
LIN {X 0,Y 378.871,Z 1208.975,A -85,B 0,C 180,E1 17911.143,E2 17911.143} C_VEL
LIN {X 0,Y 379.589,Z 1203.702,A -85,B 0,C 180,E1 17920.353,E2 17920.353} C_VEL
LIN {X 0,Y 383.362,Z 1186.533,A -85,B 0,C 180,E1 17931.275,E2 17931.275} C_VEL
LIN {X 0,Y 395.382,Z 1154.031,A -85,B 0,C 180,E1 17942.593,E2 17942.593} C_VEL
LIN {X 0,Y 416.076,Z 1106.843,A -85,B 0,C 180,E1 17952.613,E2 17952.613} C_VEL
LIN {X 0,Y 423.338,Z 1090.632,A -85,B 0,C 180,E1 17955.125,E2 17955.125} C_VEL
LIN {X 0,Y 427.014,Z 1068.712,A -85,B 0,C 180,E1 17958.862,E2 17958.862} C_VEL
LIN {X 0,Y 452.831,Z 1004.363,A -85,B 0,C 180,E1 17965.126,E2 17965.126} C_VEL
LIN {X 0,Y 474.174,Z 932.167,A -85,B 0,C 180,E1 17969.587,E2 17969.587} C_VEL
LIN {X 0,Y 457.567,Z 888.42,A -85,B 0,C 180,E1 17977.161,E2 17977.161} C_VEL
LIN {X 0,Y 440.091,Z 855.517,A -85,B 0,C 180,E1 17985.932,E2 17985.932} C_VEL
LIN {X 0,Y 429.013,Z 837.027,A -85,B 0,C 180,E1 17994.695,E2 17994.695} C_VEL
LIN {X 0,Y 425.738,Z 830.37,A -85,B 0,C 180,E1 18003.084,E2 18003.084} C_VEL
LIN {X 0,Y 430.627,Z 840.943,A -85,B 0,C 180,E1 18013.441,E2 18013.441} C_VEL
LIN {X 0,Y 443.101,Z 861.553,A -85,B 0,C 180,E1 18022.142,E2 18022.142} C_VEL
LIN {X 0,Y 459.91,Z 896.215,A -85,B 0,C 180,E1 18030.492,E2 18030.492} C_VEL
LIN {X 0,Y 473.151,Z 934.902,A -85,B 0,C 180,E1 18036.988,E2 18036.988} C_VEL
LIN {X 0,Y 449.84,Z 1007.32,A -85,B 0,C 180,E1 18041.59,E2 18041.59} C_VEL
LIN {X 0,Y 423.949,Z 1070.526,A -85,B 0,C 180,E1 18048.228,E2 18048.228} C_VEL
LIN {X 0,Y 399.773,Z 1122.661,A -85,B 0,C 180,E1 18056.96,E2 18056.96} C_VEL
LIN {X 0,Y 381.909,Z 1162.866,A -85,B 0,C 180,E1 18067.842,E2 18067.842} C_VEL
LIN {X 0,Y 373.201,Z 1188.074,A -85,B 0,C 180,E1 18079.467,E2 18079.467} C_VEL
LIN {X 0,Y 371.047,Z 1198.445,A -85,B 0,C 180,E1 18088.832,E2 18088.832} C_VEL
LIN {X 0,Y 370.667,Z 1200.638,A -85,B 0,C 180,E1 18098.236,E2 18098.236} C_VEL
LIN {X 0,Y 372.143,Z 1193.19,A -85,B 0,C 180,E1 18109.029,E2 18109.029} C_VEL
LIN {X 0,Y 378.739,Z 1172.472,A -85,B 0,C 180,E1 18120.865,E2 18120.865} C_VEL
LIN {X 0,Y 395.318,Z 1135.945,A -85,B 0,C 180,E1 18132.594,E2 18132.594} C_VEL
LIN {X 0,Y 420.453,Z 1086.381,A -85,B 0,C 180,E1 18142.217,E2 18142.217} C_VEL
LIN {X 0,Y 448.301,Z 1026.909,A -85,B 0,C 180,E1 18149.377,E2 18149.377} C_VEL
LIN {X 0,Y 474.879,Z 957.313,A -85,B 0,C 180,E1 18154.462,E2 18154.462} C_VEL
LIN {X 0,Y 481.099,Z 935.94,A -85,B 0,C 180,E1 18155.652,E2 18155.652} C_VEL
LIN {X 0,Y 469.24,Z 900.508,A -85,B 0,C 180,E1 18163.067,E2 18163.067} C_VEL
LIN {X 0,Y 457.715,Z 874.657,A -85,B 0,C 180,E1 18171.884,E2 18171.884} C_VEL
LIN {X 0,Y 452.27,Z 865.547,A -85,B 0,C 180,E1 18179.981,E2 18179.981} C_VEL
LIN {X 0,Y 452.992,Z 867.289,A -85,B 0,C 180,E1 18187.763,E2 18187.763} C_VEL
LIN {X 0,Y 458.325,Z 877.217,A -85,B 0,C 180,E1 18194.536,E2 18194.536} C_VEL
LIN {X 0,Y 469.943,Z 901.209,A -85,B 0,C 180,E1 18202.769,E2 18202.769} C_VEL
LIN {X 0,Y 482.02,Z 935.826,A -85,B 0,C 180,E1 18209.931,E2 18209.931} C_VEL
LIN {X 0,Y 457.905,Z 1008.176,A -85,B 0,C 180,E1 18214.419,E2 18214.419} C_VEL
LIN {X 0,Y 430.3,Z 1071.049,A -85,B 0,C 180,E1 18220.677,E2 18220.677} C_VEL
LIN {X 0,Y 403.663,Z 1124.62,A -85,B 0,C 180,E1 18229.248,E2 18229.248} C_VEL
LIN {X 0,Y 384.13,Z 1165.54,A -85,B 0,C 180,E1 18239.775,E2 18239.775} C_VEL
LIN {X 0,Y 374.119,Z 1192.424,A -85,B 0,C 180,E1 18251.075,E2 18251.075} C_VEL
LIN {X 0,Y 371.389,Z 1205.831,A -85,B 0,C 180,E1 18261.78,E2 18261.78} C_VEL
LIN {X 0,Y 370.878,Z 1208.883,A -85,B 0,C 180,E1 18271.168,E2 18271.168} C_VEL
LIN {X 0,Y 371.602,Z 1203.581,A -85,B 0,C 180,E1 18280.578,E2 18280.578} C_VEL
LIN {X 0,Y 375.59,Z 1186.631,A -85,B 0,C 180,E1 18291.605,E2 18291.605} C_VEL
LIN {X 0,Y 387.832,Z 1154.851,A -85,B 0,C 180,E1 18302.96,E2 18302.96} C_VEL
LIN {X 0,Y 408.965,Z 1108.627,A -85,B 0,C 180,E1 18313.058,E2 18313.058} C_VEL
LIN {X 0,Y 427.014,Z 1068.712,A -85,B 0,C 180,E1 18318.862,E2 18318.862} C_VEL
LIN {X 0,Y 431.634,Z 1045.024,A -85,B 0,C 180,E1 18322.337,E2 18322.337} C_VEL
LIN {X 0,Y 456.56,Z 979.722,A -85,B 0,C 180,E1 18327.656,E2 18327.656} C_VEL
LIN {X 0,Y 468.885,Z 936.108,A -85,B 0,C 180,E1 18330.194,E2 18330.194} C_VEL
LIN {X 0,Y 453.526,Z 894.051,A -85,B 0,C 180,E1 18337.729,E2 18337.729} C_VEL
LIN {X 0,Y 437.379,Z 862.454,A -85,B 0,C 180,E1 18346.354,E2 18346.354} C_VEL
LIN {X 0,Y 427.15,Z 844.637,A -85,B 0,C 180,E1 18355.055,E2 18355.055} C_VEL
LIN {X 0,Y 424.252,Z 838.202,A -85,B 0,C 180,E1 18363.095,E2 18363.095} C_VEL
LIN {X 0,Y 428.994,Z 848.853,A -85,B 0,C 180,E1 18373.377,E2 18373.377} C_VEL
LIN {X 0,Y 441.194,Z 869.865,A -85,B 0,C 180,E1 18382.234,E2 18382.234} C_VEL
LIN {X 0,Y 457.228,Z 905.418,A -85,B 0,C 180,E1 18390.69,E2 18390.69} C_VEL
LIN {X 0,Y 467.742,Z 938.78,A -85,B 0,C 180,E1 18396.352,E2 18396.352} C_VEL
LIN {X 0,Y 444.085,Z 1009.504,A -85,B 0,C 180,E1 18400.933,E2 18400.933} C_VEL
LIN {X 0,Y 417.952,Z 1071.147,A -85,B 0,C 180,E1 18407.49,E2 18407.49} C_VEL
LIN {X 0,Y 393.155,Z 1122.649,A -85,B 0,C 180,E1 18416.205,E2 18416.205} C_VEL
LIN {X 0,Y 374.993,Z 1161.526,A -85,B 0,C 180,E1 18426.782,E2 18426.782} C_VEL
LIN {X 0,Y 366.012,Z 1186.42,A -85,B 0,C 180,E1 18438.048,E2 18438.048} C_VEL
LIN {X 0,Y 363.051,Z 1198.602,A -85,B 0,C 180,E1 18448.807,E2 18448.807} C_VEL
LIN {X 0,Y 362.656,Z 1200.713,A -85,B 0,C 180,E1 18458.419,E2 18458.419} C_VEL
LIN {X 0,Y 364.257,Z 1193.232,A -85,B 0,C 180,E1 18469.394,E2 18469.394} C_VEL
LIN {X 0,Y 371.323,Z 1172.315,A -85,B 0,C 180,E1 18481.567,E2 18481.567} C_VEL
LIN {X 0,Y 389.044,Z 1135.433,A -85,B 0,C 180,E1 18493.524,E2 18493.524} C_VEL
LIN {X 0,Y 414.777,Z 1086.766,A -85,B 0,C 180,E1 18503.046,E2 18503.046} C_VEL
LIN {X 0,Y 443.723,Z 1026.962,A -85,B 0,C 180,E1 18510.263,E2 18510.263} C_VEL
LIN {X 0,Y 470.449,Z 959.043,A -85,B 0,C 180,E1 18515.238,E2 18515.238} C_VEL
LIN {X 0,Y 475.937,Z 939.006,A -85,B 0,C 180,E1 18516.503,E2 18516.503} C_VEL
LIN {X 0,Y 465.075,Z 905.488,A -85,B 0,C 180,E1 18523.886,E2 18523.886} C_VEL
LIN {X 0,Y 454.821,Z 881.815,A -85,B 0,C 180,E1 18532.405,E2 18532.405} C_VEL
LIN {X 0,Y 450.263,Z 873.3,A -85,B 0,C 180,E1 18539.981,E2 18539.981} C_VEL
LIN {X 0,Y 450.953,Z 875.043,A -85,B 0,C 180,E1 18547.798,E2 18547.798} C_VEL
LIN {X 0,Y 456.593,Z 886.304,A -85,B 0,C 180,E1 18555.085,E2 18555.085} C_VEL
LIN {X 0,Y 468.296,Z 912.174,A -85,B 0,C 180,E1 18563.533,E2 18563.533} C_VEL
LIN {X 0,Y 476.946,Z 941.726,A -85,B 0,C 180,E1 18569.441,E2 18569.441} C_VEL
LIN {X 0,Y 451.39,Z 1013.365,A -85,B 0,C 180,E1 18573.951,E2 18573.951} C_VEL
LIN {X 0,Y 422.412,Z 1076.38,A -85,B 0,C 180,E1 18580.49,E2 18580.49} C_VEL
LIN {X 0,Y 394.649,Z 1130.016,A -85,B 0,C 180,E1 18589.573,E2 18589.573} C_VEL
LIN {X 0,Y 374.777,Z 1170.24,A -85,B 0,C 180,E1 18600.741,E2 18600.741} C_VEL
LIN {X 0,Y 365.754,Z 1194.914,A -85,B 0,C 180,E1 18612.25,E2 18612.25} C_VEL
LIN {X 0,Y 363.168,Z 1207.349,A -85,B 0,C 180,E1 18624.004,E2 18624.004} C_VEL
LIN {X 0,Y 363.157,Z 1208.301,A -85,B 0,C 180,E1 18633.588,E2 18633.588} C_VEL
LIN {X 0,Y 364.386,Z 1199.237,A -85,B 0,C 180,E1 18644.456,E2 18644.456} C_VEL
LIN {X 0,Y 371.945,Z 1176.023,A -85,B 0,C 180,E1 18656.523,E2 18656.523} C_VEL
LIN {X 0,Y 388.428,Z 1138.15,A -85,B 0,C 180,E1 18667.849,E2 18667.849} C_VEL
LIN {X 0,Y 412.896,Z 1087,A -85,B 0,C 180,E1 18677.214,E2 18677.214} C_VEL
LIN {X 0,Y 431.634,Z 1045.024,A -85,B 0,C 180,E1 18682.337,E2 18682.337} C_VEL
LIN {X 0,Y 436.848,Z 1019.89,A -85,B 0,C 180,E1 18685.573,E2 18685.573} C_VEL
LIN {X 0,Y 461.961,Z 948.053,A -85,B 0,C 180,E1 18690.323,E2 18690.323} C_VEL
LIN {X 0,Y 463.176,Z 938.597,A -85,B 0,C 180,E1 18691.059,E2 18691.059} C_VEL
LIN {X 0,Y 448.399,Z 897.142,A -85,B 0,C 180,E1 18698.837,E2 18698.837} C_VEL
LIN {X 0,Y 432.835,Z 865.448,A -85,B 0,C 180,E1 18708.139,E2 18708.139} C_VEL
LIN {X 0,Y 424.31,Z 850.983,A -85,B 0,C 180,E1 18716.804,E2 18716.804} C_VEL
LIN {X 0,Y 422.739,Z 846.053,A -85,B 0,C 180,E1 18723.106,E2 18723.106} C_VEL
LIN {X 0,Y 427.115,Z 856.73,A -85,B 0,C 180,E1 18733.368,E2 18733.368} C_VEL
LIN {X 0,Y 438.551,Z 877.66,A -85,B 0,C 180,E1 18742.13,E2 18742.13} C_VEL
LIN {X 0,Y 453.551,Z 912.907,A -85,B 0,C 180,E1 18750.566,E2 18750.566} C_VEL
LIN {X 0,Y 462.193,Z 943.381,A -85,B 0,C 180,E1 18755.738,E2 18755.738} C_VEL
LIN {X 0,Y 437.332,Z 1014.368,A -85,B 0,C 180,E1 18760.48,E2 18760.48} C_VEL
LIN {X 0,Y 410.273,Z 1075.587,A -85,B 0,C 180,E1 18767.245,E2 18767.245} C_VEL
LIN {X 0,Y 384.863,Z 1126.457,A -85,B 0,C 180,E1 18776.265,E2 18776.265} C_VEL
LIN {X 0,Y 366.212,Z 1165.194,A -85,B 0,C 180,E1 18787.482,E2 18787.482} C_VEL
LIN {X 0,Y 357.434,Z 1188.548,A -85,B 0,C 180,E1 18798.997,E2 18798.997} C_VEL
LIN {X 0,Y 355.06,Z 1198.756,A -85,B 0,C 180,E1 18808.78,E2 18808.78} C_VEL
LIN {X 0,Y 354.648,Z 1200.787,A -85,B 0,C 180,E1 18818.611,E2 18818.611} C_VEL
LIN {X 0,Y 356.405,Z 1193.297,A -85,B 0,C 180,E1 18829.758,E2 18829.758} C_VEL
LIN {X 0,Y 363.772,Z 1172.566,A -85,B 0,C 180,E1 18842.112,E2 18842.112} C_VEL
LIN {X 0,Y 381.917,Z 1136.798,A -85,B 0,C 180,E1 18854.021,E2 18854.021} C_VEL
LIN {X 0,Y 408.647,Z 1088.205,A -85,B 0,C 180,E1 18863.738,E2 18863.738} C_VEL
LIN {X 0,Y 438.579,Z 1028.556,A -85,B 0,C 180,E1 18871.026,E2 18871.026} C_VEL
LIN {X 0,Y 466.47,Z 959.635,A -85,B 0,C 180,E1 18876.096,E2 18876.096} C_VEL
LIN {X 0,Y 471.015,Z 942.834,A -85,B 0,C 180,E1 18877.245,E2 18877.245} C_VEL
LIN {X 0,Y 460.461,Z 909.122,A -85,B 0,C 180,E1 18885.079,E2 18885.079} C_VEL
LIN {X 0,Y 452.423,Z 889.391,A -85,B 0,C 180,E1 18892.516,E2 18892.516} C_VEL
LIN {X 0,Y 448.042,Z 880.996,A -85,B 0,C 180,E1 18899.981,E2 18899.981} C_VEL
LIN {X 0,Y 448.764,Z 882.788,A -85,B 0,C 180,E1 18907.873,E2 18907.873} C_VEL
LIN {X 0,Y 455.178,Z 895.788,A -85,B 0,C 180,E1 18915.972,E2 18915.972} C_VEL
LIN {X 0,Y 466.386,Z 924.049,A -85,B 0,C 180,E1 18924.478,E2 18924.478} C_VEL
LIN {X 0,Y 471.612,Z 947.233,A -85,B 0,C 180,E1 18928.823,E2 18928.823} C_VEL
LIN {X 0,Y 444.604,Z 1019.238,A -85,B 0,C 180,E1 18933.52,E2 18933.52} C_VEL
LIN {X 0,Y 414.948,Z 1080.925,A -85,B 0,C 180,E1 18940.194,E2 18940.194} C_VEL
LIN {X 0,Y 386.983,Z 1132.76,A -85,B 0,C 180,E1 18949.343,E2 18949.343} C_VEL
LIN {X 0,Y 366.823,Z 1171.843,A -85,B 0,C 180,E1 18960.664,E2 18960.664} C_VEL
LIN {X 0,Y 357.342,Z 1197.065,A -85,B 0,C 180,E1 18973.251,E2 18973.251} C_VEL
LIN {X 0,Y 355.188,Z 1207.276,A -85,B 0,C 180,E1 18983.869,E2 18983.869} C_VEL
LIN {X 0,Y 355.158,Z 1208.198,A -85,B 0,C 180,E1 18993.669,E2 18993.669} C_VEL
LIN {X 0,Y 356.493,Z 1199.097,A -85,B 0,C 180,E1 19004.784,E2 19004.784} C_VEL
LIN {X 0,Y 364.613,Z 1175.309,A -85,B 0,C 180,E1 19017.317,E2 19017.317} C_VEL
LIN {X 0,Y 382.237,Z 1136.78,A -85,B 0,C 180,E1 19028.893,E2 19028.893} C_VEL
LIN {X 0,Y 407.202,Z 1086.603,A -85,B 0,C 180,E1 19038.086,E2 19038.086} C_VEL
LIN {X 0,Y 434.557,Z 1025.352,A -85,B 0,C 180,E1 19045.087,E2 19045.087} C_VEL
LIN {X 0,Y 436.848,Z 1019.89,A -85,B 0,C 180,E1 19045.573,E2 19045.573} C_VEL
LIN {X 0,Y 442.605,Z 992.892,A -85,B 0,C 180,E1 19048.489,E2 19048.489} C_VEL
LIN {X 0,Y 458.154,Z 943.326,A -85,B 0,C 180,E1 19051.584,E2 19051.584} C_VEL
LIN {X 0,Y 445.013,Z 904.321,A -85,B 0,C 180,E1 19059.05,E2 19059.05} C_VEL
LIN {X 0,Y 430.487,Z 872.992,A -85,B 0,C 180,E1 19068.348,E2 19068.348} C_VEL
LIN {X 0,Y 422.369,Z 858.669,A -85,B 0,C 180,E1 19076.933,E2 19076.933} C_VEL
LIN {X 0,Y 421.145,Z 853.895,A -85,B 0,C 180,E1 19084.152,E2 19084.152} C_VEL
LIN {X 0,Y 426.904,Z 866.899,A -85,B 0,C 180,E1 19094.949,E2 19094.949} C_VEL
LIN {X 0,Y 439.539,Z 893.503,A -85,B 0,C 180,E1 19104.344,E2 19104.344} C_VEL
LIN {X 0,Y 453.464,Z 931.684,A -85,B 0,C 180,E1 19112.599,E2 19112.599} C_VEL
LIN {X 0,Y 456.622,Z 947.607,A -85,B 0,C 180,E1 19115.098,E2 19115.098} C_VEL
LIN {X 0,Y 430.925,Z 1018.036,A -85,B 0,C 180,E1 19119.936,E2 19119.936} C_VEL
LIN {X 0,Y 402.995,Z 1078.802,A -85,B 0,C 180,E1 19126.854,E2 19126.854} C_VEL
LIN {X 0,Y 377.027,Z 1128.873,A -85,B 0,C 180,E1 19136.057,E2 19136.057} C_VEL
LIN {X 0,Y 358.025,Z 1167.006,A -85,B 0,C 180,E1 19147.595,E2 19147.595} C_VEL
LIN {X 0,Y 348.945,Z 1190.522,A -85,B 0,C 180,E1 19159.993,E2 19159.993} C_VEL
LIN {X 0,Y 347.232,Z 1200.117,A -85,B 0,C 180,E1 19171.255,E2 19171.255} C_VEL
LIN {X 0,Y 346.828,Z 1200.029,A -85,B 0,C 180,E1 19181.351,E2 19181.351} C_VEL
LIN {X 0,Y 349.549,Z 1189.921,A -85,B 0,C 180,E1 19192.986,E2 19192.986} C_VEL
LIN {X 0,Y 359.208,Z 1166.25,A -85,B 0,C 180,E1 19205.463,E2 19205.463} C_VEL
LIN {X 0,Y 380.565,Z 1127.903,A -85,B 0,C 180,E1 19217.075,E2 19217.075} C_VEL
LIN {X 0,Y 409.709,Z 1076.652,A -85,B 0,C 180,E1 19226.392,E2 19226.392} C_VEL
LIN {X 0,Y 440.314,Z 1015.666,A -85,B 0,C 180,E1 19233.092,E2 19233.092} C_VEL
LIN {X 0,Y 466.325,Z 947.856,A -85,B 0,C 180,E1 19237.761,E2 19237.761} C_VEL
LIN {X 0,Y 456.711,Z 915.32,A -85,B 0,C 180,E1 19245.556,E2 19245.556} C_VEL
LIN {X 0,Y 449.162,Z 896.16,A -85,B 0,C 180,E1 19253.192,E2 19253.192} C_VEL
LIN {X 0,Y 445.712,Z 888.474,A -85,B 0,C 180,E1 19260.468,E2 19260.468} C_VEL
LIN {X 0,Y 447.056,Z 890.978,A -85,B 0,C 180,E1 19268.763,E2 19268.763} C_VEL
LIN {X 0,Y 454.489,Z 908.544,A -85,B 0,C 180,E1 19277.821,E2 19277.821} C_VEL
LIN {X 0,Y 464.641,Z 937.757,A -85,B 0,C 180,E1 19285.787,E2 19285.787} C_VEL
LIN {X 0,Y 466.75,Z 951.132,A -85,B 0,C 180,E1 19288.125,E2 19288.125} C_VEL
LIN {X 0,Y 438.954,Z 1022.207,A -85,B 0,C 180,E1 19292.862,E2 19292.862} C_VEL
LIN {X 0,Y 408.562,Z 1083.127,A -85,B 0,C 180,E1 19299.592,E2 19299.592} C_VEL
LIN {X 0,Y 379.951,Z 1134.071,A -85,B 0,C 180,E1 19308.807,E2 19308.807} C_VEL
LIN {X 0,Y 359.203,Z 1172.581,A -85,B 0,C 180,E1 19320.301,E2 19320.301} C_VEL
LIN {X 0,Y 349.517,Z 1197.042,A -85,B 0,C 180,E1 19332.864,E2 19332.864} C_VEL
LIN {X 0,Y 347.186,Z 1207.204,A -85,B 0,C 180,E1 19343.727,E2 19343.727} C_VEL
LIN {X 0,Y 347.148,Z 1208.094,A -85,B 0,C 180,E1 19353.753,E2 19353.753} C_VEL
LIN {X 0,Y 348.6,Z 1198.954,A -85,B 0,C 180,E1 19365.126,E2 19365.126} C_VEL
LIN {X 0,Y 357.048,Z 1175.321,A -85,B 0,C 180,E1 19377.848,E2 19377.848} C_VEL
LIN {X 0,Y 375.532,Z 1136.845,A -85,B 0,C 180,E1 19389.614,E2 19389.614} C_VEL
LIN {X 0,Y 402.24,Z 1084.985,A -85,B 0,C 180,E1 19399.159,E2 19399.159} C_VEL
LIN {X 0,Y 430.779,Z 1022.631,A -85,B 0,C 180,E1 19406.192,E2 19406.192} C_VEL
LIN {X 0,Y 442.605,Z 992.892,A -85,B 0,C 180,E1 19408.489,E2 19408.489} C_VEL
LIN {X 0,Y 448.237,Z 964.595,A -85,B 0,C 180,E1 19411.152,E2 19411.152} C_VEL
LIN {X 0,Y 452.751,Z 946.478,A -85,B 0,C 180,E1 19412.382,E2 19412.382} C_VEL
LIN {X 0,Y 439.774,Z 907.076,A -85,B 0,C 180,E1 19420.329,E2 19420.329} C_VEL
LIN {X 0,Y 427.2,Z 879.346,A -85,B 0,C 180,E1 19429.083,E2 19429.083} C_VEL
LIN {X 0,Y 420.218,Z 866.007,A -85,B 0,C 180,E1 19437.435,E2 19437.435} C_VEL
LIN {X 0,Y 419.279,Z 861.682,A -85,B 0,C 180,E1 19444.17,E2 19444.17} C_VEL
LIN {X 0,Y 424.585,Z 874.64,A -85,B 0,C 180,E1 19454.834,E2 19454.834} C_VEL
LIN {X 0,Y 436.324,Z 900.696,A -85,B 0,C 180,E1 19464.131,E2 19464.131} C_VEL
LIN {X 0,Y 449.214,Z 938.721,A -85,B 0,C 180,E1 19472.438,E2 19472.438} C_VEL
LIN {X 0,Y 451.16,Z 951.59,A -85,B 0,C 180,E1 19474.435,E2 19474.435} C_VEL
LIN {X 0,Y 424.288,Z 1022.29,A -85,B 0,C 180,E1 19479.43,E2 19479.43} C_VEL
LIN {X 0,Y 394.976,Z 1083.488,A -85,B 0,C 180,E1 19486.672,E2 19486.672} C_VEL
LIN {X 0,Y 368.391,Z 1132.897,A -85,B 0,C 180,E1 19496.244,E2 19496.244} C_VEL
LIN {X 0,Y 349.142,Z 1170.315,A -85,B 0,C 180,E1 19508.338,E2 19508.338} C_VEL
LIN {X 0,Y 340.531,Z 1192.264,A -85,B 0,C 180,E1 19521.037,E2 19521.037} C_VEL
LIN {X 0,Y 339.247,Z 1200.243,A -85,B 0,C 180,E1 19531.284,E2 19531.284} C_VEL
LIN {X 0,Y 338.829,Z 1200.078,A -85,B 0,C 180,E1 19541.623,E2 19541.623} C_VEL
LIN {X 0,Y 341.722,Z 1190.058,A -85,B 0,C 180,E1 19553.403,E2 19553.403} C_VEL
LIN {X 0,Y 351.966,Z 1166.512,A -85,B 0,C 180,E1 19566.111,E2 19566.111} C_VEL
LIN {X 0,Y 374.7,Z 1127.613,A -85,B 0,C 180,E1 19578.06,E2 19578.06} C_VEL
LIN {X 0,Y 404.984,Z 1076.251,A -85,B 0,C 180,E1 19587.412,E2 19587.412} C_VEL
LIN {X 0,Y 435.918,Z 1016.324,A -85,B 0,C 180,E1 19593.979,E2 19593.979} C_VEL
LIN {X 0,Y 461.476,Z 952.272,A -85,B 0,C 180,E1 19598.404,E2 19598.404} C_VEL
LIN {X 0,Y 452.605,Z 920.301,A -85,B 0,C 180,E1 19606.412,E2 19606.412} C_VEL
LIN {X 0,Y 445.832,Z 902.444,A -85,B 0,C 180,E1 19614.122,E2 19614.122} C_VEL
LIN {X 0,Y 443.145,Z 895.859,A -85,B 0,C 180,E1 19620.961,E2 19620.961} C_VEL
LIN {X 0,Y 445.059,Z 899.595,A -85,B 0,C 180,E1 19629.792,E2 19629.792} C_VEL
LIN {X 0,Y 452.789,Z 919.861,A -85,B 0,C 180,E1 19639.044,E2 19639.044} C_VEL
LIN {X 0,Y 461.952,Z 950.048,A -85,B 0,C 180,E1 19646.711,E2 19646.711} C_VEL
LIN {X 0,Y 461.208,Z 956.904,A -85,B 0,C 180,E1 19647.518,E2 19647.518} C_VEL
LIN {X 0,Y 432.201,Z 1027.577,A -85,B 0,C 180,E1 19652.4,E2 19652.4} C_VEL
LIN {X 0,Y 400.175,Z 1088.804,A -85,B 0,C 180,E1 19659.479,E2 19659.479} C_VEL
LIN {X 0,Y 370.273,Z 1139.859,A -85,B 0,C 180,E1 19669.344,E2 19669.344} C_VEL
LIN {X 0,Y 349.781,Z 1177.109,A -85,B 0,C 180,E1 19681.513,E2 19681.513} C_VEL
LIN {X 0,Y 340.762,Z 1199.522,A -85,B 0,C 180,E1 19694.51,E2 19694.51} C_VEL
LIN {X 0,Y 339.19,Z 1208.181,A -85,B 0,C 180,E1 19706.151,E2 19706.151} C_VEL
LIN {X 0,Y 339.168,Z 1206.942,A -85,B 0,C 180,E1 19716.414,E2 19716.414} C_VEL
LIN {X 0,Y 341.929,Z 1194.967,A -85,B 0,C 180,E1 19728.288,E2 19728.288} C_VEL
LIN {X 0,Y 352.309,Z 1169.031,A -85,B 0,C 180,E1 19740.866,E2 19740.866} C_VEL
LIN {X 0,Y 372.947,Z 1129.267,A -85,B 0,C 180,E1 19752.133,E2 19752.133} C_VEL
LIN {X 0,Y 400.751,Z 1076.712,A -85,B 0,C 180,E1 19761.173,E2 19761.173} C_VEL
LIN {X 0,Y 429.966,Z 1013.15,A -85,B 0,C 180,E1 19767.856,E2 19767.856} C_VEL
LIN {X 0,Y 448.237,Z 964.595,A -85,B 0,C 180,E1 19771.152,E2 19771.152} C_VEL
LIN {X 0,Y 448.76,Z 951.61,A -85,B 0,C 180,E1 19772.647,E2 19772.647} C_VEL
LIN {X 0,Y 445.265,Z 941.541,A -85,B 0,C 180,E1 19774.656,E2 19774.656} C_VEL
LIN {X 0,Y 433.063,Z 906.104,A -85,B 0,C 180,E1 19782.7,E2 19782.7} C_VEL
LIN {X 0,Y 422.094,Z 881.346,A -85,B 0,C 180,E1 19791.821,E2 19791.821} C_VEL
LIN {X 0,Y 417.446,Z 869.539,A -85,B 0,C 180,E1 19801.74,E2 19801.74} C_VEL
LIN {X 0,Y 419.505,Z 876.385,A -85,B 0,C 180,E1 19811.228,E2 19811.228} C_VEL
LIN {X 0,Y 428.593,Z 897.022,A -85,B 0,C 180,E1 19820.64,E2 19820.64} C_VEL
LIN {X 0,Y 440.837,Z 931.004,A -85,B 0,C 180,E1 19829.384,E2 19829.384} C_VEL
LIN {X 0,Y 445.872,Z 955.326,A -85,B 0,C 180,E1 19833.751,E2 19833.751} C_VEL
LIN {X 0,Y 419.085,Z 1023.383,A -85,B 0,C 180,E1 19838.615,E2 19838.615} C_VEL
LIN {X 0,Y 388.777,Z 1084.692,A -85,B 0,C 180,E1 19845.951,E2 19845.951} C_VEL
LIN {X 0,Y 361.645,Z 1133.32,A -85,B 0,C 180,E1 19855.527,E2 19855.527} C_VEL
LIN {X 0,Y 341.636,Z 1170.622,A -85,B 0,C 180,E1 19867.838,E2 19867.838} C_VEL
LIN {X 0,Y 332.602,Z 1192.466,A -85,B 0,C 180,E1 19880.821,E2 19880.821} C_VEL
LIN {X 0,Y 331.236,Z 1200.369,A -85,B 0,C 180,E1 19891.315,E2 19891.315} C_VEL
LIN {X 0,Y 330.843,Z 1200.129,A -85,B 0,C 180,E1 19901.907,E2 19901.907} C_VEL
LIN {X 0,Y 333.928,Z 1190.119,A -85,B 0,C 180,E1 19913.901,E2 19913.901} C_VEL
LIN {X 0,Y 344.964,Z 1166.466,A -85,B 0,C 180,E1 19926.919,E2 19926.919} C_VEL
LIN {X 0,Y 368.509,Z 1128.041,A -85,B 0,C 180,E1 19938.894,E2 19938.894} C_VEL
LIN {X 0,Y 400.387,Z 1075.84,A -85,B 0,C 180,E1 19948.456,E2 19948.456} C_VEL
LIN {X 0,Y 432.495,Z 1015.238,A -85,B 0,C 180,E1 19955.037,E2 19955.037} C_VEL
LIN {X 0,Y 456.431,Z 955.644,A -85,B 0,C 180,E1 19959.292,E2 19959.292} C_VEL
LIN {X 0,Y 448.572,Z 925.367,A -85,B 0,C 180,E1 19967.283,E2 19967.283} C_VEL
LIN {X 0,Y 442.642,Z 908.641,A -85,B 0,C 180,E1 19975.066,E2 19975.066} C_VEL
LIN {X 0,Y 440.594,Z 902.74,A -85,B 0,C 180,E1 19982.94,E2 19982.94} C_VEL
LIN {X 0,Y 443.489,Z 910.725,A -85,B 0,C 180,E1 19991.822,E2 19991.822} C_VEL
LIN {X 0,Y 451.353,Z 932.689,A -85,B 0,C 180,E1 20000.643,E2 20000.643} C_VEL
LIN {X 0,Y 457.507,Z 957.648,A -85,B 0,C 180,E1 20006.631,E2 20006.631} C_VEL
LIN {X 0,Y 427.888,Z 1027.957,A -85,B 0,C 180,E1 20011.478,E2 20011.478} C_VEL
LIN {X 0,Y 395.183,Z 1088.694,A -85,B 0,C 180,E1 20018.505,E2 20018.505} C_VEL
LIN {X 0,Y 364.469,Z 1139.196,A -85,B 0,C 180,E1 20028.296,E2 20028.296} C_VEL
LIN {X 0,Y 343.184,Z 1175.612,A -85,B 0,C 180,E1 20040.187,E2 20040.187} C_VEL
LIN {X 0,Y 333.504,Z 1197.916,A -85,B 0,C 180,E1 20052.805,E2 20052.805} C_VEL
LIN {X 0,Y 331.181,Z 1207.063,A -85,B 0,C 180,E1 20063.423,E2 20063.423} C_VEL
LIN {X 0,Y 331.143,Z 1207.883,A -85,B 0,C 180,E1 20073.935,E2 20073.935} C_VEL
LIN {X 0,Y 332.877,Z 1198.663,A -85,B 0,C 180,E1 20085.859,E2 20085.859} C_VEL
LIN {X 0,Y 342.255,Z 1174.892,A -85,B 0,C 180,E1 20099.165,E2 20099.165} C_VEL
LIN {X 0,Y 362.095,Z 1137.328,A -85,B 0,C 180,E1 20111.047,E2 20111.047} C_VEL
LIN {X 0,Y 389.945,Z 1086.943,A -85,B 0,C 180,E1 20120.612,E2 20120.612} C_VEL
LIN {X 0,Y 420.093,Z 1025.071,A -85,B 0,C 180,E1 20127.761,E2 20127.761} C_VEL
LIN {X 0,Y 447.418,Z 954.177,A -85,B 0,C 180,E1 20132.617,E2 20132.617} C_VEL
LIN {X 0,Y 445.265,Z 941.541,A -85,B 0,C 180,E1 20134.656,E2 20134.656} C_VEL
LIN {X 0,Y 435.516,Z 929.316,A -85,B 0,C 180,E1 20138.826,E2 20138.826} C_VEL
LIN {X 0,Y 423.865,Z 898.756,A -85,B 0,C 180,E1 20147.622,E2 20147.622} C_VEL
LIN {X 0,Y 416.528,Z 882.424,A -85,B 0,C 180,E1 20156.388,E2 20156.388} C_VEL
LIN {X 0,Y 415.246,Z 877.164,A -85,B 0,C 180,E1 20164.211,E2 20164.211} C_VEL
LIN {X 0,Y 419.54,Z 889.615,A -85,B 0,C 180,E1 20174.413,E2 20174.413} C_VEL
LIN {X 0,Y 429.25,Z 914.058,A -85,B 0,C 180,E1 20183.447,E2 20183.447} C_VEL
LIN {X 0,Y 440.253,Z 951.773,A -85,B 0,C 180,E1 20191.978,E2 20191.978} C_VEL
LIN {X 0,Y 439.902,Z 961.282,A -85,B 0,C 180,E1 20193.171,E2 20193.171} C_VEL
LIN {X 0,Y 411.74,Z 1029.542,A -85,B 0,C 180,E1 20198.263,E2 20198.263} C_VEL
LIN {X 0,Y 380.577,Z 1089.697,A -85,B 0,C 180,E1 20205.793,E2 20205.793} C_VEL
LIN {X 0,Y 352.331,Z 1138.329,A -85,B 0,C 180,E1 20215.981,E2 20215.981} C_VEL
LIN {X 0,Y 332.638,Z 1173.765,A -85,B 0,C 180,E1 20228.614,E2 20228.614} C_VEL
LIN {X 0,Y 324.365,Z 1194.195,A -85,B 0,C 180,E1 20241.941,E2 20241.941} C_VEL
LIN {X 0,Y 322.936,Z 1201.186,A -85,B 0,C 180,E1 20254.043,E2 20254.043} C_VEL
LIN {X 0,Y 323.361,Z 1198.261,A -85,B 0,C 180,E1 20265.823,E2 20265.823} C_VEL
LIN {X 0,Y 329.012,Z 1183.66,A -85,B 0,C 180,E1 20278.949,E2 20278.949} C_VEL
LIN {X 0,Y 346.617,Z 1153.07,A -85,B 0,C 180,E1 20292.702,E2 20292.702} C_VEL
LIN {X 0,Y 375.067,Z 1109.003,A -85,B 0,C 180,E1 20303.952,E2 20303.952} C_VEL
LIN {X 0,Y 408.722,Z 1053.053,A -85,B 0,C 180,E1 20312.337,E2 20312.337} C_VEL
LIN {X 0,Y 441.283,Z 987.593,A -85,B 0,C 180,E1 20318.075,E2 20318.075} C_VEL
LIN {X 0,Y 451.786,Z 960.672,A -85,B 0,C 180,E1 20319.85,E2 20319.85} C_VEL
LIN {X 0,Y 444.842,Z 931.842,A -85,B 0,C 180,E1 20327.675,E2 20327.675} C_VEL
LIN {X 0,Y 439.712,Z 916.211,A -85,B 0,C 180,E1 20335.033,E2 20335.033} C_VEL
LIN {X 0,Y 437.982,Z 910.32,A -85,B 0,C 180,E1 20342.958,E2 20342.958} C_VEL
LIN {X 0,Y 440.575,Z 918.372,A -85,B 0,C 180,E1 20351.902,E2 20351.902} C_VEL
LIN {X 0,Y 447.501,Z 939.252,A -85,B 0,C 180,E1 20360.33,E2 20360.33} C_VEL
LIN {X 0,Y 452.215,Z 963.21,A -85,B 0,C 180,E1 20365.993,E2 20365.993} C_VEL
LIN {X 0,Y 421.836,Z 1032.087,A -85,B 0,C 180,E1 20370.87,E2 20370.87} C_VEL
LIN {X 0,Y 388.906,Z 1090.888,A -85,B 0,C 180,E1 20377.846,E2 20377.846} C_VEL
LIN {X 0,Y 357.444,Z 1140.633,A -85,B 0,C 180,E1 20387.738,E2 20387.738} C_VEL
LIN {X 0,Y 335.17,Z 1177.179,A -85,B 0,C 180,E1 20400.149,E2 20400.149} C_VEL
LIN {X 0,Y 325.018,Z 1199.634,A -85,B 0,C 180,E1 20413.893,E2 20413.893} C_VEL
LIN {X 0,Y 323.164,Z 1208.041,A -85,B 0,C 180,E1 20425.96,E2 20425.96} C_VEL
LIN {X 0,Y 323.167,Z 1206.729,A -85,B 0,C 180,E1 20436.733,E2 20436.733} C_VEL
LIN {X 0,Y 326.182,Z 1194.941,A -85,B 0,C 180,E1 20448.988,E2 20448.988} C_VEL
LIN {X 0,Y 337.366,Z 1169.768,A -85,B 0,C 180,E1 20461.877,E2 20461.877} C_VEL
LIN {X 0,Y 359.776,Z 1129.968,A -85,B 0,C 180,E1 20473.641,E2 20473.641} C_VEL
LIN {X 0,Y 389.729,Z 1077.13,A -85,B 0,C 180,E1 20482.923,E2 20482.923} C_VEL
LIN {X 0,Y 420.119,Z 1014.76,A -85,B 0,C 180,E1 20489.548,E2 20489.548} C_VEL
LIN {X 0,Y 442.492,Z 955.023,A -85,B 0,C 180,E1 20493.62,E2 20493.62} C_VEL
LIN {X 0,Y 435.516,Z 929.316,A -85,B 0,C 180,E1 20498.826,E2 20498.826} C_VEL
LIN {X 0,Y 426.146,Z 919.958,A -85,B 0,C 180,E1 20503.23,E2 20503.23} C_VEL
LIN {X 0,Y 417.337,Z 897.245,A -85,B 0,C 180,E1 20511.662,E2 20511.662} C_VEL
LIN {X 0,Y 413.023,Z 884.871,A -85,B 0,C 180,E1 20522.126,E2 20522.126} C_VEL
LIN {X 0,Y 415.55,Z 894.754,A -85,B 0,C 180,E1 20532.726,E2 20532.726} C_VEL
LIN {X 0,Y 423.789,Z 915.471,A -85,B 0,C 180,E1 20541.545,E2 20541.545} C_VEL
LIN {X 0,Y 433.524,Z 948.879,A -85,B 0,C 180,E1 20549.849,E2 20549.849} C_VEL
LIN {X 0,Y 435.622,Z 962.315,A -85,B 0,C 180,E1 20552.299,E2 20552.299} C_VEL
LIN {X 0,Y 406.583,Z 1030.781,A -85,B 0,C 180,E1 20557.425,E2 20557.425} C_VEL
LIN {X 0,Y 374.821,Z 1090.21,A -85,B 0,C 180,E1 20564.931,E2 20564.931} C_VEL
LIN {X 0,Y 345.601,Z 1138.715,A -85,B 0,C 180,E1 20575.225,E2 20575.225} C_VEL
LIN {X 0,Y 325.112,Z 1174.039,A -85,B 0,C 180,E1 20588.094,E2 20588.094} C_VEL
LIN {X 0,Y 316.415,Z 1194.376,A -85,B 0,C 180,E1 20601.737,E2 20601.737} C_VEL
LIN {X 0,Y 314.903,Z 1201.286,A -85,B 0,C 180,E1 20614.146,E2 20614.146} C_VEL
LIN {X 0,Y 315.285,Z 1198.826,A -85,B 0,C 180,E1 20625.344,E2 20625.344} C_VEL
LIN {X 0,Y 320.167,Z 1186.283,A -85,B 0,C 180,E1 20637.91,E2 20637.91} C_VEL
LIN {X 0,Y 337.169,Z 1157.673,A -85,B 0,C 180,E1 20652.033,E2 20652.033} C_VEL
LIN {X 0,Y 364.924,Z 1116.383,A -85,B 0,C 180,E1 20663.5,E2 20663.5} C_VEL
LIN {X 0,Y 399.28,Z 1062.298,A -85,B 0,C 180,E1 20672.269,E2 20672.269} C_VEL
LIN {X 0,Y 433.301,Z 997.924,A -85,B 0,C 180,E1 20678.35,E2 20678.35} C_VEL
LIN {X 0,Y 447.029,Z 965.622,A -85,B 0,C 180,E1 20680.432,E2 20680.432} C_VEL
LIN {X 0,Y 440.666,Z 936.785,A -85,B 0,C 180,E1 20688.615,E2 20688.615} C_VEL
LIN {X 0,Y 436.212,Z 921.428,A -85,B 0,C 180,E1 20696.572,E2 20696.572} C_VEL
LIN {X 0,Y 435.105,Z 918.601,A -85,B 0,C 180,E1 20704.98,E2 20704.98} C_VEL
LIN {X 0,Y 438.253,Z 927.886,A -85,B 0,C 180,E1 20712.981,E2 20712.981} C_VEL
LIN {X 0,Y 444.944,Z 950.65,A -85,B 0,C 180,E1 20721.438,E2 20721.438} C_VEL
LIN {X 0,Y 447.611,Z 966.999,A -85,B 0,C 180,E1 20725.243,E2 20725.243} C_VEL
LIN {X 0,Y 415.81,Z 1036.183,A -85,B 0,C 180,E1 20730.248,E2 20730.248} C_VEL
LIN {X 0,Y 380.757,Z 1096.186,A -85,B 0,C 180,E1 20737.662,E2 20737.662} C_VEL
LIN {X 0,Y 348.377,Z 1145.089,A -85,B 0,C 180,E1 20747.985,E2 20747.985} C_VEL
LIN {X 0,Y 326.407,Z 1180.108,A -85,B 0,C 180,E1 20760.798,E2 20760.798} C_VEL
LIN {X 0,Y 316.647,Z 1200.995,A -85,B 0,C 180,E1 20774.724,E2 20774.724} C_VEL
LIN {X 0,Y 315.151,Z 1207.968,A -85,B 0,C 180,E1 20785.857,E2 20785.857} C_VEL
LIN {X 0,Y 315.163,Z 1206.62,A -85,B 0,C 180,E1 20796.905,E2 20796.905} C_VEL
LIN {X 0,Y 318.353,Z 1194.774,A -85,B 0,C 180,E1 20809.474,E2 20809.474} C_VEL
LIN {X 0,Y 330.252,Z 1169.528,A -85,B 0,C 180,E1 20822.648,E2 20822.648} C_VEL
LIN {X 0,Y 353.677,Z 1129.631,A -85,B 0,C 180,E1 20834.591,E2 20834.591} C_VEL
LIN {X 0,Y 384.651,Z 1076.766,A -85,B 0,C 180,E1 20843.914,E2 20843.914} C_VEL
LIN {X 0,Y 416.029,Z 1014.049,A -85,B 0,C 180,E1 20850.538,E2 20850.538} C_VEL
LIN {X 0,Y 437.294,Z 958.911,A -85,B 0,C 180,E1 20854.326,E2 20854.326} C_VEL
LIN {X 0,Y 427.12,Z 922.723,A -85,B 0,C 180,E1 20862.452,E2 20862.452} C_VEL
LIN {X 0,Y 426.146,Z 919.958,A -85,B 0,C 180,E1 20863.23,E2 20863.23} C_VEL
LIN {X 0,Y 417.977,Z 913.673,A -85,B 0,C 180,E1 20867.869,E2 20867.869} C_VEL
LIN {X 0,Y 411.489,Z 897.326,A -85,B 0,C 180,E1 20876.851,E2 20876.851} C_VEL
LIN {X 0,Y 410.661,Z 892.442,A -85,B 0,C 180,E1 20883.197,E2 20883.197} C_VEL
LIN {X 0,Y 413.733,Z 904.06,A -85,B 0,C 180,E1 20893.808,E2 20893.808} C_VEL
LIN {X 0,Y 421.917,Z 927.32,A -85,B 0,C 180,E1 20902.759,E2 20902.759} C_VEL
LIN {X 0,Y 430.81,Z 963.683,A -85,B 0,C 180,E1 20911.312,E2 20911.312} C_VEL
LIN {X 0,Y 400.754,Z 1033.382,A -85,B 0,C 180,E1 20916.709,E2 20916.709} C_VEL
LIN {X 0,Y 368.341,Z 1092.001,A -85,B 0,C 180,E1 20924.259,E2 20924.259} C_VEL
LIN {X 0,Y 338.935,Z 1139.096,A -85,B 0,C 180,E1 20934.438,E2 20934.438} C_VEL
LIN {X 0,Y 317.615,Z 1174.313,A -85,B 0,C 180,E1 20947.549,E2 20947.549} C_VEL
LIN {X 0,Y 308.459,Z 1194.55,A -85,B 0,C 180,E1 20961.523,E2 20961.523} C_VEL
LIN {X 0,Y 306.88,Z 1201.386,A -85,B 0,C 180,E1 20974.255,E2 20974.255} C_VEL
LIN {X 0,Y 307.346,Z 1198.854,A -85,B 0,C 180,E1 20985.75,E2 20985.75} C_VEL
LIN {X 0,Y 313.469,Z 1184.882,A -85,B 0,C 180,E1 20999.588,E2 20999.588} C_VEL
LIN {X 0,Y 332.383,Z 1155.143,A -85,B 0,C 180,E1 21013.886,E2 21013.886} C_VEL
LIN {X 0,Y 362.815,Z 1111.734,A -85,B 0,C 180,E1 21025.497,E2 21025.497} C_VEL
LIN {X 0,Y 398.528,Z 1056.379,A -85,B 0,C 180,E1 21034.018,E2 21034.018} C_VEL
LIN {X 0,Y 432.941,Z 991.259,A -85,B 0,C 180,E1 21039.801,E2 21039.801} C_VEL
LIN {X 0,Y 442.016,Z 968.837,A -85,B 0,C 180,E1 21041.414,E2 21041.414} C_VEL
LIN {X 0,Y 436.667,Z 942.011,A -85,B 0,C 180,E1 21049.472,E2 21049.472} C_VEL
LIN {X 0,Y 433.122,Z 928.418,A -85,B 0,C 180,E1 21056.969,E2 21056.969} C_VEL
LIN {X 0,Y 432.204,Z 926.076,A -85,B 0,C 180,E1 21065.013,E2 21065.013} C_VEL
LIN {X 0,Y 435.02,Z 935.537,A -85,B 0,C 180,E1 21073.079,E2 21073.079} C_VEL
LIN {X 0,Y 441.185,Z 958.973,A -85,B 0,C 180,E1 21081.67,E2 21081.67} C_VEL
LIN {X 0,Y 442.772,Z 971.096,A -85,B 0,C 180,E1 21084.507,E2 21084.507} C_VEL
LIN {X 0,Y 409.823,Z 1039.906,A -85,B 0,C 180,E1 21089.586,E2 21089.586} C_VEL
LIN {X 0,Y 374.663,Z 1097.98,A -85,B 0,C 180,E1 21096.923,E2 21096.923} C_VEL
LIN {X 0,Y 341.134,Z 1146.677,A -85,B 0,C 180,E1 21107.476,E2 21107.476} C_VEL
LIN {X 0,Y 318.488,Z 1181.266,A -85,B 0,C 180,E1 21120.664,E2 21120.664} C_VEL
LIN {X 0,Y 308.789,Z 1200.959,A -85,B 0,C 180,E1 21134.325,E2 21134.325} C_VEL
LIN {X 0,Y 307.15,Z 1207.893,A -85,B 0,C 180,E1 21145.749,E2 21145.749} C_VEL
LIN {X 0,Y 307.162,Z 1206.507,A -85,B 0,C 180,E1 21157.086,E2 21157.086} C_VEL
LIN {X 0,Y 310.557,Z 1194.604,A -85,B 0,C 180,E1 21169.983,E2 21169.983} C_VEL
LIN {X 0,Y 323.198,Z 1169.283,A -85,B 0,C 180,E1 21183.453,E2 21183.453} C_VEL
LIN {X 0,Y 347.742,Z 1129.298,A -85,B 0,C 180,E1 21195.564,E2 21195.564} C_VEL
LIN {X 0,Y 379.77,Z 1076.313,A -85,B 0,C 180,E1 21204.938,E2 21204.938} C_VEL
LIN {X 0,Y 411.999,Z 1013.424,A -85,B 0,C 180,E1 21211.546,E2 21211.546} C_VEL
LIN {X 0,Y 432.157,Z 962.857,A -85,B 0,C 180,E1 21215.043,E2 21215.043} C_VEL
LIN {X 0,Y 422.792,Z 927.355,A -85,B 0,C 180,E1 21223.342,E2 21223.342} C_VEL
LIN {X 0,Y 417.977,Z 913.673,A -85,B 0,C 180,E1 21227.869,E2 21227.869} C_VEL
LIN {X 0,Y 411.161,Z 910.92,A -85,B 0,C 180,E1 21232.688,E2 21232.688} C_VEL
LIN {X 0,Y 408.077,Z 900.088,A -85,B 0,C 180,E1 21243.218,E2 21243.218} C_VEL
LIN {X 0,Y 410.979,Z 911.926,A -85,B 0,C 180,E1 21253.903,E2 21253.903} C_VEL
LIN {X 0,Y 418.505,Z 935.676,A -85,B 0,C 180,E1 21262.955,E2 21262.955} C_VEL
LIN {X 0,Y 425.575,Z 968.74,A -85,B 0,C 180,E1 21270.773,E2 21270.773} C_VEL
LIN {X 0,Y 395.422,Z 1035.178,A -85,B 0,C 180,E1 21275.895,E2 21275.895} C_VEL
LIN {X 0,Y 362.325,Z 1093.146,A -85,B 0,C 180,E1 21283.452,E2 21283.452} C_VEL
LIN {X 0,Y 331.569,Z 1140.605,A -85,B 0,C 180,E1 21293.955,E2 21293.955} C_VEL
LIN {X 0,Y 310.149,Z 1174.583,A -85,B 0,C 180,E1 21306.978,E2 21306.978} C_VEL
LIN {X 0,Y 300.541,Z 1194.721,A -85,B 0,C 180,E1 21321.298,E2 21321.298} C_VEL
LIN {X 0,Y 298.848,Z 1201.486,A -85,B 0,C 180,E1 21334.37,E2 21334.37} C_VEL
LIN {X 0,Y 299.399,Z 1198.883,A -85,B 0,C 180,E1 21346.18,E2 21346.18} C_VEL
LIN {X 0,Y 306.062,Z 1184.873,A -85,B 0,C 180,E1 21360.334,E2 21360.334} C_VEL
LIN {X 0,Y 325.128,Z 1156.441,A -85,B 0,C 180,E1 21374.427,E2 21374.427} C_VEL
LIN {X 0,Y 356.165,Z 1113.999,A -85,B 0,C 180,E1 21386.132,E2 21386.132} C_VEL
LIN {X 0,Y 392.942,Z 1059.11,A -85,B 0,C 180,E1 21394.764,E2 21394.764} C_VEL
LIN {X 0,Y 427.87,Z 995.391,A -85,B 0,C 180,E1 21400.533,E2 21400.533} C_VEL
LIN {X 0,Y 437.252,Z 973.519,A -85,B 0,C 180,E1 21402.078,E2 21402.078} C_VEL
LIN {X 0,Y 432.65,Z 947.154,A -85,B 0,C 180,E1 21410.393,E2 21410.393} C_VEL
LIN {X 0,Y 429.321,Z 934.148,A -85,B 0,C 180,E1 21418.968,E2 21418.968} C_VEL
LIN {X 0,Y 429.063,Z 933.486,A -85,B 0,C 180,E1 21425.05,E2 21425.05} C_VEL
LIN {X 0,Y 431.729,Z 943.173,A -85,B 0,C 180,E1 21433.181,E2 21433.181} C_VEL
LIN {X 0,Y 437.19,Z 966.435,A -85,B 0,C 180,E1 21441.648,E2 21441.648} C_VEL
LIN {X 0,Y 437.267,Z 976.951,A -85,B 0,C 180,E1 21443.858,E2 21443.858} C_VEL
LIN {X 0,Y 403.183,Z 1044.878,A -85,B 0,C 180,E1 21449.025,E2 21449.025} C_VEL
LIN {X 0,Y 366.07,Z 1103.565,A -85,B 0,C 180,E1 21456.809,E2 21456.809} C_VEL
LIN {X 0,Y 333.32,Z 1149.146,A -85,B 0,C 180,E1 21467.211,E2 21467.211} C_VEL
LIN {X 0,Y 310.297,Z 1182.83,A -85,B 0,C 180,E1 21480.739,E2 21480.739} C_VEL
LIN {X 0,Y 300.41,Z 1202.141,A -85,B 0,C 180,E1 21495.376,E2 21495.376} C_VEL
LIN {X 0,Y 298.992,Z 1208.17,A -85,B 0,C 180,E1 21508.543,E2 21508.543} C_VEL
LIN {X 0,Y 299.544,Z 1204.644,A -85,B 0,C 180,E1 21520.202,E2 21520.202} C_VEL
LIN {X 0,Y 304.788,Z 1189.846,A -85,B 0,C 180,E1 21533.737,E2 21533.737} C_VEL
LIN {X 0,Y 322.129,Z 1159.854,A -85,B 0,C 180,E1 21547.728,E2 21547.728} C_VEL
LIN {X 0,Y 350.121,Z 1116.384,A -85,B 0,C 180,E1 21559.28,E2 21559.28} C_VEL
LIN {X 0,Y 383.313,Z 1061.235,A -85,B 0,C 180,E1 21567.849,E2 21567.849} C_VEL
LIN {X 0,Y 415.508,Z 996.358,A -85,B 0,C 180,E1 21573.795,E2 21573.795} C_VEL
LIN {X 0,Y 426.929,Z 966.199,A -85,B 0,C 180,E1 21575.906,E2 21575.906} C_VEL
LIN {X 0,Y 418.383,Z 932.147,A -85,B 0,C 180,E1 21584.243,E2 21584.243} C_VEL
LIN {X 0,Y 411.161,Z 910.92,A -85,B 0,C 180,E1 21592.688,E2 21592.688} C_VEL
LIN {X 0,Y 405.897,Z 911.772,A -85,B 0,C 180,E1 21597.641,E2 21597.641} C_VEL
LIN {X 0,Y 405.5,Z 907.719,A -85,B 0,C 180,E1 21603.238,E2 21603.238} C_VEL
LIN {X 0,Y 408.013,Z 919.766,A -85,B 0,C 180,E1 21614.006,E2 21614.006} C_VEL
LIN {X 0,Y 414.584,Z 942.203,A -85,B 0,C 180,E1 21622.615,E2 21622.615} C_VEL
LIN {X 0,Y 420.118,Z 973.239,A -85,B 0,C 180,E1 21630.057,E2 21630.057} C_VEL
LIN {X 0,Y 388.954,Z 1039.222,A -85,B 0,C 180,E1 21635.288,E2 21635.288} C_VEL
LIN {X 0,Y 354.362,Z 1097.343,A -85,B 0,C 180,E1 21643.144,E2 21643.144} C_VEL
LIN {X 0,Y 322.891,Z 1144.097,A -85,B 0,C 180,E1 21654.056,E2 21654.056} C_VEL
LIN {X 0,Y 301.086,Z 1177.473,A -85,B 0,C 180,E1 21667.81,E2 21667.81} C_VEL
LIN {X 0,Y 292.246,Z 1196.079,A -85,B 0,C 180,E1 21682.551,E2 21682.551} C_VEL
LIN {X 0,Y 290.816,Z 1201.586,A -85,B 0,C 180,E1 21694.49,E2 21694.49} C_VEL
LIN {X 0,Y 291.466,Z 1198.912,A -85,B 0,C 180,E1 21706.633,E2 21706.633} C_VEL
LIN {X 0,Y 298.805,Z 1184.661,A -85,B 0,C 180,E1 21721.254,E2 21721.254} C_VEL
LIN {X 0,Y 320.087,Z 1154.603,A -85,B 0,C 180,E1 21736.127,E2 21736.127} C_VEL
LIN {X 0,Y 352.381,Z 1112.35,A -85,B 0,C 180,E1 21747.572,E2 21747.572} C_VEL
LIN {X 0,Y 390.004,Z 1057.565,A -85,B 0,C 180,E1 21756.037,E2 21756.037} C_VEL
LIN {X 0,Y 426.004,Z 992.896,A -85,B 0,C 180,E1 21761.716,E2 21761.716} C_VEL
LIN {X 0,Y 432.585,Z 978.692,A -85,B 0,C 180,E1 21762.638,E2 21762.638} C_VEL
LIN {X 0,Y 428.741,Z 953.474,A -85,B 0,C 180,E1 21770.819,E2 21770.819} C_VEL
LIN {X 0,Y 426.076,Z 941.483,A -85,B 0,C 180,E1 21778.96,E2 21778.96} C_VEL
LIN {X 0,Y 425.822,Z 940.838,A -85,B 0,C 180,E1 21785.089,E2 21785.089} C_VEL
LIN {X 0,Y 428.303,Z 950.749,A -85,B 0,C 180,E1 21793.288,E2 21793.288} C_VEL
LIN {X 0,Y 433.042,Z 974.51,A -85,B 0,C 180,E1 21801.868,E2 21801.868} C_VEL
LIN {X 0,Y 432.219,Z 981.911,A -85,B 0,C 180,E1 21803.148,E2 21803.148} C_VEL
LIN {X 0,Y 397.318,Z 1048.621,A -85,B 0,C 180,E1 21808.332,E2 21808.332} C_VEL
LIN {X 0,Y 358.936,Z 1107.017,A -85,B 0,C 180,E1 21816.317,E2 21816.317} C_VEL
LIN {X 0,Y 324.595,Z 1152.953,A -85,B 0,C 180,E1 21827.353,E2 21827.353} C_VEL
LIN {X 0,Y 301.179,Z 1185.985,A -85,B 0,C 180,E1 21841.747,E2 21841.747} C_VEL
LIN {X 0,Y 292.041,Z 1203.321,A -85,B 0,C 180,E1 21856.482,E2 21856.482} C_VEL
LIN {X 0,Y 291.015,Z 1208.09,A -85,B 0,C 180,E1 21868.503,E2 21868.503} C_VEL
LIN {X 0,Y 291.56,Z 1204.52,A -85,B 0,C 180,E1 21880.484,E2 21880.484} C_VEL
LIN {X 0,Y 297.317,Z 1189.488,A -85,B 0,C 180,E1 21894.486,E2 21894.486} C_VEL
LIN {X 0,Y 315.535,Z 1159.585,A -85,B 0,C 180,E1 21908.661,E2 21908.661} C_VEL
LIN {X 0,Y 344.99,Z 1115.582,A -85,B 0,C 180,E1 21920.424,E2 21920.424} C_VEL
LIN {X 0,Y 379.864,Z 1059.048,A -85,B 0,C 180,E1 21929.12,E2 21929.12} C_VEL
LIN {X 0,Y 412.291,Z 994.756,A -85,B 0,C 180,E1 21934.897,E2 21934.897} C_VEL
LIN {X 0,Y 421.733,Z 969.822,A -85,B 0,C 180,E1 21936.715,E2 21936.715} C_VEL
LIN {X 0,Y 414.389,Z 938.243,A -85,B 0,C 180,E1 21944.716,E2 21944.716} C_VEL
LIN {X 0,Y 407.598,Z 917.017,A -85,B 0,C 180,E1 21953.611,E2 21953.611} C_VEL
LIN {X 0,Y 405.897,Z 911.772,A -85,B 0,C 180,E1 21957.641,E2 21957.641} C_VEL
LIN {X 0,Y 402.6,Z 915.424,A -85,B 0,C 180,E1 21962.661,E2 21962.661} C_VEL
LIN {X 0,Y 404.452,Z 925.617,A -85,B 0,C 180,E1 21973.026,E2 21973.026} C_VEL
LIN {X 0,Y 410.175,Z 946.85,A -85,B 0,C 180,E1 21981.727,E2 21981.727} C_VEL
LIN {X 0,Y 415.256,Z 976.452,A -85,B 0,C 180,E1 21989.247,E2 21989.247} C_VEL
LIN {X 0,Y 383.158,Z 1042.137,A -85,B 0,C 180,E1 21994.547,E2 21994.547} C_VEL
LIN {X 0,Y 347.646,Z 1099.725,A -85,B 0,C 180,E1 22002.509,E2 22002.509} C_VEL
LIN {X 0,Y 315.588,Z 1145.533,A -85,B 0,C 180,E1 22013.518,E2 22013.518} C_VEL
LIN {X 0,Y 293.606,Z 1177.741,A -85,B 0,C 180,E1 22027.214,E2 22027.214} C_VEL
LIN {X 0,Y 284.287,Z 1196.249,A -85,B 0,C 180,E1 22042.341,E2 22042.341} C_VEL
LIN {X 0,Y 282.786,Z 1201.686,A -85,B 0,C 180,E1 22054.618,E2 22054.618} C_VEL
LIN {X 0,Y 283.545,Z 1198.942,A -85,B 0,C 180,E1 22067.111,E2 22067.111} C_VEL
LIN {X 0,Y 291.628,Z 1184.39,A -85,B 0,C 180,E1 22082.267,E2 22082.267} C_VEL
LIN {X 0,Y 314.175,Z 1154.354,A -85,B 0,C 180,E1 22097.296,E2 22097.296} C_VEL
LIN {X 0,Y 348.712,Z 1110.856,A -85,B 0,C 180,E1 22109.014,E2 22109.014} C_VEL
LIN {X 0,Y 387.575,Z 1055.543,A -85,B 0,C 180,E1 22117.379,E2 22117.379} C_VEL
LIN {X 0,Y 424.132,Z 990.753,A -85,B 0,C 180,E1 22122.893,E2 22122.893} C_VEL
LIN {X 0,Y 427.686,Z 982.155,A -85,B 0,C 180,E1 22123.674,E2 22123.674} C_VEL
LIN {X 0,Y 424.492,Z 957.582,A -85,B 0,C 180,E1 22132.279,E2 22132.279} C_VEL
LIN {X 0,Y 422.727,Z 948.77,A -85,B 0,C 180,E1 22138.951,E2 22138.951} C_VEL
LIN {X 0,Y 422.525,Z 948.177,A -85,B 0,C 180,E1 22145.129,E2 22145.129} C_VEL
LIN {X 0,Y 424.668,Z 958.255,A -85,B 0,C 180,E1 22153.404,E2 22153.404} C_VEL
LIN {X 0,Y 428.66,Z 981.596,A -85,B 0,C 180,E1 22161.79,E2 22161.79} C_VEL
LIN {X 0,Y 424.328,Z 992.598,A -85,B 0,C 180,E1 22162.787,E2 22162.787} C_VEL
LIN {X 0,Y 387.565,Z 1058.437,A -85,B 0,C 180,E1 22168.305,E2 22168.305} C_VEL
LIN {X 0,Y 349.068,Z 1113.848,A -85,B 0,C 180,E1 22176.51,E2 22176.51} C_VEL
LIN {X 0,Y 314.512,Z 1158.134,A -85,B 0,C 180,E1 22188.118,E2 22188.118} C_VEL
LIN {X 0,Y 292.354,Z 1188.21,A -85,B 0,C 180,E1 22202.44,E2 22202.44} C_VEL
LIN {X 0,Y 284.151,Z 1203.283,A -85,B 0,C 180,E1 22216.1,E2 22216.1} C_VEL
LIN {X 0,Y 283.011,Z 1208.009,A -85,B 0,C 180,E1 22228.46,E2 22228.46} C_VEL
LIN {X 0,Y 283.593,Z 1204.396,A -85,B 0,C 180,E1 22240.782,E2 22240.782} C_VEL
LIN {X 0,Y 290.135,Z 1188.725,A -85,B 0,C 180,E1 22255.539,E2 22255.539} C_VEL
LIN {X 0,Y 310.473,Z 1157.322,A -85,B 0,C 180,E1 22270.324,E2 22270.324} C_VEL
LIN {X 0,Y 341.484,Z 1112.664,A -85,B 0,C 180,E1 22282.015,E2 22282.015} C_VEL
LIN {X 0,Y 376.57,Z 1056.927,A -85,B 0,C 180,E1 22290.405,E2 22290.405} C_VEL
LIN {X 0,Y 410.027,Z 991.445,A -85,B 0,C 180,E1 22296.12,E2 22296.12} C_VEL
LIN {X 0,Y 416.579,Z 973.422,A -85,B 0,C 180,E1 22297.545,E2 22297.545} C_VEL
LIN {X 0,Y 409.686,Z 941.587,A -85,B 0,C 180,E1 22306.096,E2 22306.096} C_VEL
LIN {X 0,Y 404.113,Z 922.952,A -85,B 0,C 180,E1 22314.637,E2 22314.637} C_VEL
LIN {X 0,Y 402.6,Z 915.424,A -85,B 0,C 180,E1 22322.661,E2 22322.661} C_VEL
LIN {X 0,Y 399.425,Z 926.337,A -85,B 0,C 180,E1 22327.484,E2 22327.484} C_VEL
LIN {X 0,Y 402.957,Z 939.805,A -85,B 0,C 180,E1 22336.421,E2 22336.421} C_VEL
LIN {X 0,Y 408.379,Z 965.975,A -85,B 0,C 180,E1 22345.016,E2 22345.016} C_VEL
LIN {X 0,Y 409.4,Z 982.161,A -85,B 0,C 180,E1 22348.576,E2 22348.576} C_VEL
LIN {X 0,Y 376.14,Z 1047.268,A -85,B 0,C 180,E1 22354.009,E2 22354.009} C_VEL
LIN {X 0,Y 338.82,Z 1105.06,A -85,B 0,C 180,E1 22362.403,E2 22362.403} C_VEL
LIN {X 0,Y 306.833,Z 1148.973,A -85,B 0,C 180,E1 22373.63,E2 22373.63} C_VEL
LIN {X 0,Y 284.51,Z 1180.521,A -85,B 0,C 180,E1 22388.098,E2 22388.098} C_VEL
LIN {X 0,Y 276.34,Z 1196.418,A -85,B 0,C 180,E1 22402.119,E2 22402.119} C_VEL
LIN {X 0,Y 274.769,Z 1201.785,A -85,B 0,C 180,E1 22414.753,E2 22414.753} C_VEL
LIN {X 0,Y 275.651,Z 1198.973,A -85,B 0,C 180,E1 22427.617,E2 22427.617} C_VEL
LIN {X 0,Y 284.364,Z 1184.393,A -85,B 0,C 180,E1 22443.14,E2 22443.14} C_VEL
LIN {X 0,Y 307.77,Z 1154.837,A -85,B 0,C 180,E1 22458.253,E2 22458.253} C_VEL
LIN {X 0,Y 343.263,Z 1111.944,A -85,B 0,C 180,E1 22469.971,E2 22469.971} C_VEL
LIN {X 0,Y 383.352,Z 1056.646,A -85,B 0,C 180,E1 22478.383,E2 22478.383} C_VEL
LIN {X 0,Y 421.091,Z 991.361,A -85,B 0,C 180,E1 22483.907,E2 22483.907} C_VEL
LIN {X 0,Y 422.818,Z 984.931,A -85,B 0,C 180,E1 22484.903,E2 22484.903} C_VEL
LIN {X 0,Y 420.334,Z 962.499,A -85,B 0,C 180,E1 22493.588,E2 22493.588} C_VEL
LIN {X 0,Y 418.911,Z 954.992,A -85,B 0,C 180,E1 22501.017,E2 22501.017} C_VEL
LIN {X 0,Y 419.717,Z 958.828,A -85,B 0,C 180,E1 22509.339,E2 22509.339} C_VEL
LIN {X 0,Y 422.719,Z 976.747,A -85,B 0,C 180,E1 22518.064,E2 22518.064} C_VEL
LIN {X 0,Y 423.367,Z 988.822,A -85,B 0,C 180,E1 22521.5,E2 22521.5} C_VEL
LIN {X 0,Y 385.991,Z 1055.288,A -85,B 0,C 180,E1 22526.842,E2 22526.842} C_VEL
LIN {X 0,Y 346.026,Z 1111.647,A -85,B 0,C 180,E1 22534.924,E2 22534.924} C_VEL
LIN {X 0,Y 309.249,Z 1157.024,A -85,B 0,C 180,E1 22546.64,E2 22546.64} C_VEL
LIN {X 0,Y 284.6,Z 1188.811,A -85,B 0,C 180,E1 22562.066,E2 22562.066} C_VEL
LIN {X 0,Y 276.252,Z 1203.245,A -85,B 0,C 180,E1 22575.694,E2 22575.694} C_VEL
LIN {X 0,Y 275.022,Z 1207.929,A -85,B 0,C 180,E1 22588.416,E2 22588.416} C_VEL
LIN {X 0,Y 275.621,Z 1204.271,A -85,B 0,C 180,E1 22601.098,E2 22601.098} C_VEL
LIN {X 0,Y 282.7,Z 1188.532,A -85,B 0,C 180,E1 22616.261,E2 22616.261} C_VEL
LIN {X 0,Y 304.104,Z 1157.047,A -85,B 0,C 180,E1 22631.35,E2 22631.35} C_VEL
LIN {X 0,Y 336.314,Z 1112.287,A -85,B 0,C 180,E1 22643.158,E2 22643.158} C_VEL
LIN {X 0,Y 373.069,Z 1055.461,A -85,B 0,C 180,E1 22651.638,E2 22651.638} C_VEL
LIN {X 0,Y 406.871,Z 990.457,A -85,B 0,C 180,E1 22657.207,E2 22657.207} C_VEL
LIN {X 0,Y 411.627,Z 978.316,A -85,B 0,C 180,E1 22658.12,E2 22658.12} C_VEL
LIN {X 0,Y 405.843,Z 947.967,A -85,B 0,C 180,E1 22666.513,E2 22666.513} C_VEL
LIN {X 0,Y 400.745,Z 928.898,A -85,B 0,C 180,E1 22675.68,E2 22675.68} C_VEL
LIN {X 0,Y 399.721,Z 922.78,A -85,B 0,C 180,E1 22683.285,E2 22683.285} C_VEL
LIN {X 0,Y 399.425,Z 926.337,A -85,B 0,C 180,E1 22687.484,E2 22687.484} C_VEL
LIN {X 0,Y 397.539,Z 939.316,A -85,B 0,C 180,E1 22692.258,E2 22692.258} C_VEL
LIN {X 0,Y 401.91,Z 959.635,A -85,B 0,C 180,E1 22701.034,E2 22701.034} C_VEL
LIN {X 0,Y 404.688,Z 985.062,A -85,B 0,C 180,E1 22707.727,E2 22707.727} C_VEL
LIN {X 0,Y 370.254,Z 1050.189,A -85,B 0,C 180,E1 22713.241,E2 22713.241} C_VEL
LIN {X 0,Y 332.331,Z 1106.945,A -85,B 0,C 180,E1 22721.657,E2 22721.657} C_VEL
LIN {X 0,Y 298.775,Z 1151.223,A -85,B 0,C 180,E1 22733.394,E2 22733.394} C_VEL
LIN {X 0,Y 276.197,Z 1181.887,A -85,B 0,C 180,E1 22748.252,E2 22748.252} C_VEL
LIN {X 0,Y 268.165,Z 1197.775,A -85,B 0,C 180,E1 22763.511,E2 22763.511} C_VEL
LIN {X 0,Y 266.711,Z 1201.92,A -85,B 0,C 180,E1 22775.228,E2 22775.228} C_VEL
LIN {X 0,Y 267.763,Z 1199.004,A -85,B 0,C 180,E1 22788.154,E2 22788.154} C_VEL
LIN {X 0,Y 277.171,Z 1184.326,A -85,B 0,C 180,E1 22804.116,E2 22804.116} C_VEL
LIN {X 0,Y 302.003,Z 1154.661,A -85,B 0,C 180,E1 22819.494,E2 22819.494} C_VEL
LIN {X 0,Y 339.439,Z 1111.097,A -85,B 0,C 180,E1 22831.352,E2 22831.352} C_VEL
LIN {X 0,Y 380.308,Z 1056.198,A -85,B 0,C 180,E1 22839.571,E2 22839.571} C_VEL
LIN {X 0,Y 418.16,Z 991.357,A -85,B 0,C 180,E1 22845.115,E2 22845.115} C_VEL
LIN {X 0,Y 416.44,Z 969.734,A -85,B 0,C 180,E1 22853.528,E2 22853.528} C_VEL
LIN {X 0,Y 415.348,Z 962.15,A -85,B 0,C 180,E1 22861.025,E2 22861.025} C_VEL
LIN {X 0,Y 416.068,Z 966.189,A -85,B 0,C 180,E1 22869.421,E2 22869.421} C_VEL
LIN {X 0,Y 418.49,Z 983.576,A -85,B 0,C 180,E1 22877.922,E2 22877.922} C_VEL
LIN {X 0,Y 418.339,Z 993.645,A -85,B 0,C 180,E1 22880.746,E2 22880.746} C_VEL
LIN {X 0,Y 380.055,Z 1059.093,A -85,B 0,C 180,E1 22886.126,E2 22886.126} C_VEL
LIN {X 0,Y 339.42,Z 1114.238,A -85,B 0,C 180,E1 22894.248,E2 22894.248} C_VEL
LIN {X 0,Y 303.163,Z 1157.118,A -85,B 0,C 180,E1 22905.543,E2 22905.543} C_VEL
LIN {X 0,Y 277.28,Z 1188.825,A -85,B 0,C 180,E1 22921.261,E2 22921.261} C_VEL
LIN {X 0,Y 268.359,Z 1203.209,A -85,B 0,C 180,E1 22935.264,E2 22935.264} C_VEL
LIN {X 0,Y 267.017,Z 1207.848,A -85,B 0,C 180,E1 22948.368,E2 22948.368} C_VEL
LIN {X 0,Y 267.663,Z 1204.145,A -85,B 0,C 180,E1 22961.432,E2 22961.432} C_VEL
LIN {X 0,Y 275.286,Z 1188.338,A -85,B 0,C 180,E1 22977.025,E2 22977.025} C_VEL
LIN {X 0,Y 297.825,Z 1156.734,A -85,B 0,C 180,E1 22992.439,E2 22992.439} C_VEL
LIN {X 0,Y 331.035,Z 1112.32,A -85,B 0,C 180,E1 23004.24,E2 23004.24} C_VEL
LIN {X 0,Y 368.928,Z 1055.343,A -85,B 0,C 180,E1 23012.735,E2 23012.735} C_VEL
LIN {X 0,Y 403.633,Z 989.963,A -85,B 0,C 180,E1 23018.277,E2 23018.277} C_VEL
LIN {X 0,Y 406.397,Z 980.895,A -85,B 0,C 180,E1 23019.255,E2 23019.255} C_VEL
LIN {X 0,Y 401.165,Z 951.227,A -85,B 0,C 180,E1 23028.019,E2 23028.019} C_VEL
LIN {X 0,Y 397.126,Z 935.025,A -85,B 0,C 180,E1 23036.737,E2 23036.737} C_VEL
LIN {X 0,Y 396.705,Z 930.258,A -85,B 0,C 180,E1 23043.31,E2 23043.31} C_VEL
LIN {X 0,Y 397.539,Z 939.316,A -85,B 0,C 180,E1 23052.258,E2 23052.258} C_VEL
LIN {X 0,Y 395.892,Z 955.641,A -85,B 0,C 180,E1 23056.839,E2 23056.839} C_VEL
LIN {X 0,Y 399.621,Z 981.912,A -85,B 0,C 180,E1 23065.303,E2 23065.303} C_VEL
LIN {X 0,Y 399.141,Z 989.892,A -85,B 0,C 180,E1 23066.979,E2 23066.979} C_VEL
LIN {X 0,Y 363.484,Z 1054.647,A -85,B 0,C 180,E1 23072.628,E2 23072.628} C_VEL
LIN {X 0,Y 324.606,Z 1110.549,A -85,B 0,C 180,E1 23081.232,E2 23081.232} C_VEL
LIN {X 0,Y 290.733,Z 1153.471,A -85,B 0,C 180,E1 23093.147,E2 23093.147} C_VEL
LIN {X 0,Y 267.889,Z 1183.25,A -85,B 0,C 180,E1 23108.416,E2 23108.416} C_VEL
LIN {X 0,Y 260.178,Z 1198.067,A -85,B 0,C 180,E1 23123.497,E2 23123.497} C_VEL
LIN {X 0,Y 258.755,Z 1201.984,A -85,B 0,C 180,E1 23135.048,E2 23135.048} C_VEL
LIN {X 0,Y 260.374,Z 1198.276,A -85,B 0,C 180,E1 23150.252,E2 23150.252} C_VEL
LIN {X 0,Y 271.805,Z 1181.933,A -85,B 0,C 180,E1 23166.859,E2 23166.859} C_VEL
LIN {X 0,Y 299.955,Z 1150.613,A -85,B 0,C 180,E1 23182.201,E2 23182.201} C_VEL
LIN {X 0,Y 339.639,Z 1105.707,A -85,B 0,C 180,E1 23193.651,E2 23193.651} C_VEL
LIN {X 0,Y 382.021,Z 1049.094,A -85,B 0,C 180,E1 23201.486,E2 23201.486} C_VEL
LIN {X 0,Y 413.458,Z 995.978,A -85,B 0,C 180,E1 23205.873,E2 23205.873} C_VEL
LIN {X 0,Y 412.424,Z 976.635,A -85,B 0,C 180,E1 23213.644,E2 23213.644} C_VEL
LIN {X 0,Y 411.592,Z 969.196,A -85,B 0,C 180,E1 23221.035,E2 23221.035} C_VEL
LIN {X 0,Y 412.118,Z 973.393,A -85,B 0,C 180,E1 23229.512,E2 23229.512} C_VEL
LIN {X 0,Y 414.07,Z 991.163,A -85,B 0,C 180,E1 23238.12,E2 23238.12} C_VEL
LIN {X 0,Y 413.459,Z 998.322,A -85,B 0,C 180,E1 23239.964,E2 23239.964} C_VEL
LIN {X 0,Y 374.518,Z 1062.41,A -85,B 0,C 180,E1 23245.336,E2 23245.336} C_VEL
LIN {X 0,Y 332.449,Z 1117.322,A -85,B 0,C 180,E1 23253.64,E2 23253.64} C_VEL
LIN {X 0,Y 295.557,Z 1159.152,A -85,B 0,C 180,E1 23265.125,E2 23265.125} C_VEL
LIN {X 0,Y 269.893,Z 1188.998,A -85,B 0,C 180,E1 23280.525,E2 23280.525} C_VEL
LIN {X 0,Y 260.49,Z 1203.173,A -85,B 0,C 180,E1 23294.808,E2 23294.808} C_VEL
LIN {X 0,Y 259.028,Z 1207.768,A -85,B 0,C 180,E1 23308.318,E2 23308.318} C_VEL
LIN {X 0,Y 259.713,Z 1204.019,A -85,B 0,C 180,E1 23321.787,E2 23321.787} C_VEL
LIN {X 0,Y 267.93,Z 1188.143,A -85,B 0,C 180,E1 23337.831,E2 23337.831} C_VEL
LIN {X 0,Y 291.239,Z 1156.942,A -85,B 0,C 180,E1 23353.384,E2 23353.384} C_VEL
LIN {X 0,Y 326.011,Z 1112.174,A -85,B 0,C 180,E1 23365.393,E2 23365.393} C_VEL
LIN {X 0,Y 364.475,Z 1055.885,A -85,B 0,C 180,E1 23373.793,E2 23373.793} C_VEL
LIN {X 0,Y 400.414,Z 989.669,A -85,B 0,C 180,E1 23379.36,E2 23379.36} C_VEL
LIN {X 0,Y 400.255,Z 975.834,A -85,B 0,C 180,E1 23382.453,E2 23382.453} C_VEL
LIN {X 0,Y 395.937,Z 951.882,A -85,B 0,C 180,E1 23390.915,E2 23390.915} C_VEL
LIN {X 0,Y 393.467,Z 938.171,A -85,B 0,C 180,E1 23401.127,E2 23401.127} C_VEL
LIN {X 0,Y 393.3,Z 942.401,A -85,B 0,C 180,E1 23409.014,E2 23409.014} C_VEL
LIN {X 0,Y 395.892,Z 955.641,A -85,B 0,C 180,E1 23416.839,E2 23416.839} C_VEL
LIN {X 0,Y 393.64,Z 974.873,A -85,B 0,C 180,E1 23421.194,E2 23421.194} C_VEL
LIN {X 0,Y 394.245,Z 993.504,A -85,B 0,C 180,E1 23426.131,E2 23426.131} C_VEL
LIN {X 0,Y 357.758,Z 1057.544,A -85,B 0,C 180,E1 23431.815,E2 23431.815} C_VEL
LIN {X 0,Y 317.621,Z 1113.199,A -85,B 0,C 180,E1 23440.587,E2 23440.587} C_VEL
LIN {X 0,Y 281.931,Z 1156.637,A -85,B 0,C 180,E1 23453.232,E2 23453.232} C_VEL
LIN {X 0,Y 258.811,Z 1185.775,A -85,B 0,C 180,E1 23469.451,E2 23469.451} C_VEL
LIN {X 0,Y 251.91,Z 1198.972,A -85,B 0,C 180,E1 23484.824,E2 23484.824} C_VEL
LIN {X 0,Y 250.742,Z 1202.083,A -85,B 0,C 180,E1 23495.21,E2 23495.21} C_VEL
LIN {X 0,Y 252.046,Z 1199.068,A -85,B 0,C 180,E1 23509.329,E2 23509.329} C_VEL
LIN {X 0,Y 263.241,Z 1183.93,A -85,B 0,C 180,E1 23526.432,E2 23526.432} C_VEL
LIN {X 0,Y 292.403,Z 1152.802,A -85,B 0,C 180,E1 23542.674,E2 23542.674} C_VEL
LIN {X 0,Y 332.958,Z 1108.778,A -85,B 0,C 180,E1 23554.326,E2 23554.326} C_VEL
LIN {X 0,Y 376.455,Z 1052.831,A -85,B 0,C 180,E1 23562.269,E2 23562.269} C_VEL
LIN {X 0,Y 408.753,Z 999.993,A -85,B 0,C 180,E1 23566.84,E2 23566.84} C_VEL
LIN {X 0,Y 408.209,Z 982.188,A -85,B 0,C 180,E1 23574.648,E2 23574.648} C_VEL
LIN {X 0,Y 407.813,Z 975.74,A -85,B 0,C 180,E1 23583.177,E2 23583.177} C_VEL
LIN {X 0,Y 408.506,Z 983.902,A -85,B 0,C 180,E1 23591.762,E2 23591.762} C_VEL
LIN {X 0,Y 409.243,Z 1001.835,A -85,B 0,C 180,E1 23599.098,E2 23599.098} C_VEL
LIN {X 0,Y 369.361,Z 1065.272,A -85,B 0,C 180,E1 23604.471,E2 23604.471} C_VEL
LIN {X 0,Y 325.507,Z 1120.339,A -85,B 0,C 180,E1 23613.003,E2 23613.003} C_VEL
LIN {X 0,Y 286.426,Z 1162.834,A -85,B 0,C 180,E1 23625.348,E2 23625.348} C_VEL
LIN {X 0,Y 260.04,Z 1192.249,A -85,B 0,C 180,E1 23642.185,E2 23642.185} C_VEL
LIN {X 0,Y 251.7,Z 1204.991,A -85,B 0,C 180,E1 23657.822,E2 23657.822} C_VEL
LIN {X 0,Y 250.965,Z 1207.475,A -85,B 0,C 180,E1 23671.726,E2 23671.726} C_VEL
LIN {X 0,Y 252.672,Z 1201.551,A -85,B 0,C 180,E1 23685.664,E2 23685.664} C_VEL
LIN {X 0,Y 265.146,Z 1181.557,A -85,B 0,C 180,E1 23702.905,E2 23702.905} C_VEL
LIN {X 0,Y 292.839,Z 1147.118,A -85,B 0,C 180,E1 23717.836,E2 23717.836} C_VEL
LIN {X 0,Y 331.045,Z 1098.836,A -85,B 0,C 180,E1 23729.014,E2 23729.014} C_VEL
LIN {X 0,Y 370.422,Z 1039.703,A -85,B 0,C 180,E1 23736.601,E2 23736.601} C_VEL
LIN {X 0,Y 396.472,Z 990.417,A -85,B 0,C 180,E1 23740.52,E2 23740.52} C_VEL
LIN {X 0,Y 393.125,Z 963.772,A -85,B 0,C 180,E1 23748.899,E2 23748.899} C_VEL
LIN {X 0,Y 390.239,Z 948.641,A -85,B 0,C 180,E1 23757.795,E2 23757.795} C_VEL
LIN {X 0,Y 390.177,Z 945.021,A -85,B 0,C 180,E1 23763.365,E2 23763.365} C_VEL
LIN {X 0,Y 391.096,Z 957.047,A -85,B 0,C 180,E1 23774.051,E2 23774.051} C_VEL
LIN {X 0,Y 393.64,Z 974.873,A -85,B 0,C 180,E1 23781.194,E2 23781.194} C_VEL
LIN {X 0,Y 389.795,Z 990.703,A -85,B 0,C 180,E1 23783.772,E2 23783.772} C_VEL
LIN {X 0,Y 388.387,Z 999.195,A -85,B 0,C 180,E1 23785.4,E2 23785.4} C_VEL
LIN {X 0,Y 351.003,Z 1062.141,A -85,B 0,C 180,E1 23791.174,E2 23791.174} C_VEL
LIN {X 0,Y 310.342,Z 1116.236,A -85,B 0,C 180,E1 23800.004,E2 23800.004} C_VEL
LIN {X 0,Y 274.626,Z 1157.918,A -85,B 0,C 180,E1 23812.603,E2 23812.603} C_VEL
LIN {X 0,Y 251.288,Z 1185.959,A -85,B 0,C 180,E1 23828.765,E2 23828.765} C_VEL
LIN {X 0,Y 243.944,Z 1199.115,A -85,B 0,C 180,E1 23844.655,E2 23844.655} C_VEL
LIN {X 0,Y 242.705,Z 1202.183,A -85,B 0,C 180,E1 23855.383,E2 23855.383} C_VEL
LIN {X 0,Y 244.242,Z 1199.101,A -85,B 0,C 180,E1 23869.973,E2 23869.973} C_VEL
LIN {X 0,Y 256.049,Z 1184.174,A -85,B 0,C 180,E1 23887.346,E2 23887.346} C_VEL
LIN {X 0,Y 286.552,Z 1153.285,A -85,B 0,C 180,E1 23903.814,E2 23903.814} C_VEL
LIN {X 0,Y 329.299,Z 1108.49,A -85,B 0,C 180,E1 23915.684,E2 23915.684} C_VEL
LIN {X 0,Y 373.632,Z 1052.824,A -85,B 0,C 180,E1 23923.47,E2 23923.47} C_VEL
LIN {X 0,Y 403.924,Z 1005.163,A -85,B 0,C 180,E1 23927.434,E2 23927.434} C_VEL
LIN {X 0,Y 403.841,Z 987.688,A -85,B 0,C 180,E1 23935.67,E2 23935.67} C_VEL
LIN {X 0,Y 403.922,Z 982.74,A -85,B 0,C 180,E1 23943.208,E2 23943.208} C_VEL
LIN {X 0,Y 404.215,Z 991.013,A -85,B 0,C 180,E1 23951.889,E2 23951.889} C_VEL
LIN {X 0,Y 404.315,Z 1006.407,A -85,B 0,C 180,E1 23958.29,E2 23958.29} C_VEL
LIN {X 0,Y 362.956,Z 1069.641,A -85,B 0,C 180,E1 23963.782,E2 23963.782} C_VEL
LIN {X 0,Y 318.411,Z 1123.344,A -85,B 0,C 180,E1 23972.38,E2 23972.38} C_VEL
LIN {X 0,Y 278.345,Z 1165.069,A -85,B 0,C 180,E1 23985.074,E2 23985.074} C_VEL
LIN {X 0,Y 252.617,Z 1192.377,A -85,B 0,C 180,E1 24001.424,E2 24001.424} C_VEL
LIN {X 0,Y 243.758,Z 1204.941,A -85,B 0,C 180,E1 24017.418,E2 24017.418} C_VEL
LIN {X 0,Y 242.965,Z 1207.38,A -85,B 0,C 180,E1 24031.783,E2 24031.783} C_VEL
LIN {X 0,Y 244.879,Z 1201.282,A -85,B 0,C 180,E1 24046.362,E2 24046.362} C_VEL
LIN {X 0,Y 258.12,Z 1181.336,A -85,B 0,C 180,E1 24063.92,E2 24063.92} C_VEL
LIN {X 0,Y 287.604,Z 1146.346,A -85,B 0,C 180,E1 24079.241,E2 24079.241} C_VEL
LIN {X 0,Y 327.172,Z 1097.942,A -85,B 0,C 180,E1 24090.359,E2 24090.359} C_VEL
LIN {X 0,Y 367.41,Z 1038.789,A -85,B 0,C 180,E1 24097.829,E2 24097.829} C_VEL
LIN {X 0,Y 391.467,Z 994.814,A -85,B 0,C 180,E1 24101.262,E2 24101.262} C_VEL
LIN {X 0,Y 388.745,Z 968.724,A -85,B 0,C 180,E1 24109.91,E2 24109.91} C_VEL
LIN {X 0,Y 386.498,Z 954.853,A -85,B 0,C 180,E1 24118.898,E2 24118.898} C_VEL
LIN {X 0,Y 386.664,Z 952.286,A -85,B 0,C 180,E1 24123.396,E2 24123.396} C_VEL
LIN {X 0,Y 387.311,Z 963.85,A -85,B 0,C 180,E1 24133.779,E2 24133.779} C_VEL
LIN {X 0,Y 389.533,Z 985.812,A -85,B 0,C 180,E1 24142.333,E2 24142.333} C_VEL
LIN {X 0,Y 389.795,Z 990.703,A -85,B 0,C 180,E1 24143.772,E2 24143.772} C_VEL
LIN {X 0,Y 385.887,Z 999.832,A -85,B 0,C 180,E1 24144.63,E2 24144.63} C_VEL
LIN {X 0,Y 379.259,Z 1010.453,A -85,B 0,C 180,E1 24145.062,E2 24145.062} C_VEL
LIN {X 0,Y 339.573,Z 1072.943,A -85,B 0,C 180,E1 24151.349,E2 24151.349} C_VEL
LIN {X 0,Y 297.921,Z 1124.995,A -85,B 0,C 180,E1 24160.792,E2 24160.792} C_VEL
LIN {X 0,Y 262.641,Z 1164.158,A -85,B 0,C 180,E1 24174.215,E2 24174.215} C_VEL
LIN {X 0,Y 242.276,Z 1188.088,A -85,B 0,C 180,E1 24189.869,E2 24189.869} C_VEL
LIN {X 0,Y 235.99,Z 1199.258,A -85,B 0,C 180,E1 24204.474,E2 24204.474} C_VEL
LIN {X 0,Y 234.679,Z 1202.282,A -85,B 0,C 180,E1 24215.568,E2 24215.568} C_VEL
LIN {X 0,Y 236.783,Z 1198.695,A -85,B 0,C 180,E1 24231.639,E2 24231.639} C_VEL
LIN {X 0,Y 250.319,Z 1182.909,A -85,B 0,C 180,E1 24249.508,E2 24249.508} C_VEL
LIN {X 0,Y 282.7,Z 1151.974,A -85,B 0,C 180,E1 24265.672,E2 24265.672} C_VEL
LIN {X 0,Y 326.81,Z 1107.166,A -85,B 0,C 180,E1 24277.261,E2 24277.261} C_VEL
LIN {X 0,Y 372.183,Z 1051.209,A -85,B 0,C 180,E1 24284.841,E2 24284.841} C_VEL
LIN {X 0,Y 399.196,Z 1009.158,A -85,B 0,C 180,E1 24288.471,E2 24288.471} C_VEL
LIN {X 0,Y 399.574,Z 994.628,A -85,B 0,C 180,E1 24295.624,E2 24295.624} C_VEL
LIN {X 0,Y 399.718,Z 989.59,A -85,B 0,C 180,E1 24303.241,E2 24303.241} C_VEL
LIN {X 0,Y 399.911,Z 998.149,A -85,B 0,C 180,E1 24312.019,E2 24312.019} C_VEL
LIN {X 0,Y 399.217,Z 1011.419,A -85,B 0,C 180,E1 24317.492,E2 24317.492} C_VEL
LIN {X 0,Y 357.027,Z 1073.409,A -85,B 0,C 180,E1 24322.99,E2 24322.99} C_VEL
LIN {X 0,Y 311.721,Z 1125.945,A -85,B 0,C 180,E1 24331.635,E2 24331.635} C_VEL
LIN {X 0,Y 270.347,Z 1167.22,A -85,B 0,C 180,E1 24344.743,E2 24344.743} C_VEL
LIN {X 0,Y 243.697,Z 1194.18,A -85,B 0,C 180,E1 24362.174,E2 24362.174} C_VEL
LIN {X 0,Y 235.837,Z 1204.891,A -85,B 0,C 180,E1 24376.989,E2 24376.989} C_VEL
LIN {X 0,Y 234.988,Z 1207.285,A -85,B 0,C 180,E1 24391.844,E2 24391.844} C_VEL
LIN {X 0,Y 236.995,Z 1201.262,A -85,B 0,C 180,E1 24406.729,E2 24406.729} C_VEL
LIN {X 0,Y 250.113,Z 1182.488,A -85,B 0,C 180,E1 24424.108,E2 24424.108} C_VEL
LIN {X 0,Y 279.926,Z 1148.575,A -85,B 0,C 180,E1 24439.712,E2 24439.712} C_VEL
LIN {X 0,Y 320.45,Z 1100.839,A -85,B 0,C 180,E1 24451.093,E2 24451.093} C_VEL
LIN {X 0,Y 362.089,Z 1041.769,A -85,B 0,C 180,E1 24458.715,E2 24458.715} C_VEL
LIN {X 0,Y 386.504,Z 998.066,A -85,B 0,C 180,E1 24462.326,E2 24462.326} C_VEL
LIN {X 0,Y 384.37,Z 973.644,A -85,B 0,C 180,E1 24470.941,E2 24470.941} C_VEL
LIN {X 0,Y 382.907,Z 961.058,A -85,B 0,C 180,E1 24480.023,E2 24480.023} C_VEL
LIN {X 0,Y 382.516,Z 961.298,A -85,B 0,C 180,E1 24485.712,E2 24485.712} C_VEL
LIN {X 0,Y 383.528,Z 973.21,A -85,B 0,C 180,E1 24494.92,E2 24494.92} C_VEL
LIN {X 0,Y 385.015,Z 996.777,A -85,B 0,C 180,E1 24503.446,E2 24503.446} C_VEL
LIN {X 0,Y 382.829,Z 1003.96,A -85,B 0,C 180,E1 24504.609,E2 24504.609} C_VEL
LIN {X 0,Y 379.259,Z 1010.453,A -85,B 0,C 180,E1 24505.062,E2 24505.062} C_VEL
LIN {X 0,Y 365.069,Z 1029.671,A -85,B 0,C 180,E1 24505.416,E2 24505.416} C_VEL
LIN {X 0,Y 323.686,Z 1088.902,A -85,B 0,C 180,E1 24512.393,E2 24512.393} C_VEL
LIN {X 0,Y 280.699,Z 1138.548,A -85,B 0,C 180,E1 24523.177,E2 24523.177} C_VEL
LIN {X 0,Y 246.914,Z 1174.346,A -85,B 0,C 180,E1 24538.537,E2 24538.537} C_VEL
LIN {X 0,Y 230.188,Z 1194.977,A -85,B 0,C 180,E1 24556.675,E2 24556.675} C_VEL
LIN {X 0,Y 227.079,Z 1201.963,A -85,B 0,C 180,E1 24571.919,E2 24571.919} C_VEL
LIN {X 0,Y 227.449,Z 1200.83,A -85,B 0,C 180,E1 24587.465,E2 24587.465} C_VEL
LIN {X 0,Y 237.421,Z 1189.26,A -85,B 0,C 180,E1 24605.096,E2 24605.096} C_VEL
LIN {X 0,Y 266.548,Z 1162.17,A -85,B 0,C 180,E1 24622.934,E2 24622.934} C_VEL
LIN {X 0,Y 309.668,Z 1121.385,A -85,B 0,C 180,E1 24635.743,E2 24635.743} C_VEL
LIN {X 0,Y 356.339,Z 1068.708,A -85,B 0,C 180,E1 24644.232,E2 24644.232} C_VEL
LIN {X 0,Y 393.978,Z 1015.339,A -85,B 0,C 180,E1 24648.984,E2 24648.984} C_VEL
LIN {X 0,Y 395.22,Z 1001.506,A -85,B 0,C 180,E1 24655.576,E2 24655.576} C_VEL
LIN {X 0,Y 395.508,Z 996.429,A -85,B 0,C 180,E1 24663.276,E2 24663.276} C_VEL
LIN {X 0,Y 395.413,Z 1005.16,A -85,B 0,C 180,E1 24672.158,E2 24672.158} C_VEL
LIN {X 0,Y 394.367,Z 1016.157,A -85,B 0,C 180,E1 24676.658,E2 24676.658} C_VEL
LIN {X 0,Y 350.088,Z 1078.606,A -85,B 0,C 180,E1 24682.356,E2 24682.356} C_VEL
LIN {X 0,Y 303.394,Z 1130.303,A -85,B 0,C 180,E1 24691.252,E2 24691.252} C_VEL
LIN {X 0,Y 261.554,Z 1170.135,A -85,B 0,C 180,E1 24704.739,E2 24704.739} C_VEL
LIN {X 0,Y 234.739,Z 1196.054,A -85,B 0,C 180,E1 24723.108,E2 24723.108} C_VEL
LIN {X 0,Y 227.287,Z 1206.192,A -85,B 0,C 180,E1 24740.393,E2 24740.393} C_VEL
LIN {X 0,Y 226.98,Z 1207.189,A -85,B 0,C 180,E1 24751.909,E2 24751.909} C_VEL
LIN {X 0,Y 229.178,Z 1201.117,A -85,B 0,C 180,E1 24767.318,E2 24767.318} C_VEL
LIN {X 0,Y 243.179,Z 1182.265,A -85,B 0,C 180,E1 24785.221,E2 24785.221} C_VEL
LIN {X 0,Y 274.723,Z 1148.042,A -85,B 0,C 180,E1 24801.135,E2 24801.135} C_VEL
LIN {X 0,Y 316.472,Z 1100.42,A -85,B 0,C 180,E1 24812.425,E2 24812.425} C_VEL
LIN {X 0,Y 359.153,Z 1041.203,A -85,B 0,C 180,E1 24819.952,E2 24819.952} C_VEL
LIN {X 0,Y 381.602,Z 1002.794,A -85,B 0,C 180,E1 24823.009,E2 24823.009} C_VEL
LIN {X 0,Y 380.057,Z 978.682,A -85,B 0,C 180,E1 24831.993,E2 24831.993} C_VEL
LIN {X 0,Y 379.4,Z 967.165,A -85,B 0,C 180,E1 24841.168,E2 24841.168} C_VEL
LIN {X 0,Y 378.767,Z 971.441,A -85,B 0,C 180,E1 24849.241,E2 24849.241} C_VEL
LIN {X 0,Y 379.864,Z 987.268,A -85,B 0,C 180,E1 24857.971,E2 24857.971} C_VEL
LIN {X 0,Y 379.57,Z 1004.71,A -85,B 0,C 180,E1 24863.512,E2 24863.512} C_VEL
LIN {X 0,Y 365.069,Z 1029.671,A -85,B 0,C 180,E1 24865.416,E2 24865.416} C_VEL
LIN {X 0,Y 344.047,Z 1056.813,A -85,B 0,C 180,E1 24866.879,E2 24866.879} C_VEL
LIN {X 0,Y 299.468,Z 1112.776,A -85,B 0,C 180,E1 24875.384,E2 24875.384} C_VEL
LIN {X 0,Y 259.301,Z 1155.152,A -85,B 0,C 180,E1 24887.742,E2 24887.742} C_VEL
LIN {X 0,Y 230.766,Z 1184.429,A -85,B 0,C 180,E1 24904.72,E2 24904.72} C_VEL
LIN {X 0,Y 220.848,Z 1197.583,A -85,B 0,C 180,E1 24920.121,E2 24920.121} C_VEL
LIN {X 0,Y 218.626,Z 1202.48,A -85,B 0,C 180,E1 24935.978,E2 24935.978} C_VEL
LIN {X 0,Y 220.917,Z 1199.203,A -85,B 0,C 180,E1 24952.188,E2 24952.188} C_VEL
LIN {X 0,Y 235.9,Z 1183.951,A -85,B 0,C 180,E1 24971.224,E2 24971.224} C_VEL
LIN {X 0,Y 270.502,Z 1154.077,A -85,B 0,C 180,E1 24987.773,E2 24987.773} C_VEL
LIN {X 0,Y 317.323,Z 1109.893,A -85,B 0,C 180,E1 24999.5,E2 24999.5} C_VEL
LIN {X 0,Y 364.513,Z 1055.051,A -85,B 0,C 180,E1 25006.942,E2 25006.942} C_VEL
LIN {X 0,Y 389.609,Z 1019.177,A -85,B 0,C 180,E1 25009.887,E2 25009.887} C_VEL
LIN {X 0,Y 390.799,Z 1005.794,A -85,B 0,C 180,E1 25017.632,E2 25017.632} C_VEL
LIN {X 0,Y 390.929,Z 1004.273,A -85,B 0,C 180,E1 25025.544,E2 25025.544} C_VEL
LIN {X 0,Y 390.67,Z 1015.496,A -85,B 0,C 180,E1 25034.021,E2 25034.021} C_VEL
LIN {X 0,Y 389.093,Z 1021.378,A -85,B 0,C 180,E1 25035.847,E2 25035.847} C_VEL
LIN {X 0,Y 344.634,Z 1081.74,A -85,B 0,C 180,E1 25041.454,E2 25041.454} C_VEL
LIN {X 0,Y 295.905,Z 1133.536,A -85,B 0,C 180,E1 25050.64,E2 25050.64} C_VEL
LIN {X 0,Y 253.89,Z 1171.734,A -85,B 0,C 180,E1 25064.206,E2 25064.206} C_VEL
LIN {X 0,Y 227.389,Z 1196.039,A -85,B 0,C 180,E1 25082.165,E2 25082.165} C_VEL
LIN {X 0,Y 219.302,Z 1206.127,A -85,B 0,C 180,E1 25100.039,E2 25100.039} C_VEL
LIN {X 0,Y 218.983,Z 1207.094,A -85,B 0,C 180,E1 25111.979,E2 25111.979} C_VEL
LIN {X 0,Y 221.356,Z 1200.97,A -85,B 0,C 180,E1 25127.95,E2 25127.95} C_VEL
LIN {X 0,Y 237.11,Z 1181.2,A -85,B 0,C 180,E1 25146.964,E2 25146.964} C_VEL
LIN {X 0,Y 269.756,Z 1147.421,A -85,B 0,C 180,E1 25162.646,E2 25162.646} C_VEL
LIN {X 0,Y 312.648,Z 1099.997,A -85,B 0,C 180,E1 25173.799,E2 25173.799} C_VEL
LIN {X 0,Y 355.921,Z 1041.333,A -85,B 0,C 180,E1 25181.148,E2 25181.148} C_VEL
LIN {X 0,Y 376.605,Z 1006,A -85,B 0,C 180,E1 25184.149,E2 25184.149} C_VEL
LIN {X 0,Y 375.812,Z 983.798,A -85,B 0,C 180,E1 25193.068,E2 25193.068} C_VEL
LIN {X 0,Y 375.495,Z 974.192,A -85,B 0,C 180,E1 25201.18,E2 25201.18} C_VEL
LIN {X 0,Y 374.824,Z 978.628,A -85,B 0,C 180,E1 25209.339,E2 25209.339} C_VEL
LIN {X 0,Y 375.37,Z 995.272,A -85,B 0,C 180,E1 25218.32,E2 25218.32} C_VEL
LIN {X 0,Y 374.119,Z 1009.581,A -85,B 0,C 180,E1 25222.68,E2 25222.68} C_VEL
LIN {X 0,Y 344.047,Z 1056.813,A -85,B 0,C 180,E1 25226.879,E2 25226.879} C_VEL
LIN {X 0,Y 321.621,Z 1082.107,A -85,B 0,C 180,E1 25228.76,E2 25228.76} C_VEL
LIN {X 0,Y 277.044,Z 1131.843,A -85,B 0,C 180,E1 25238.515,E2 25238.515} C_VEL
LIN {X 0,Y 239.08,Z 1169.003,A -85,B 0,C 180,E1 25252.952,E2 25252.952} C_VEL
LIN {X 0,Y 216.776,Z 1192.282,A -85,B 0,C 180,E1 25271.657,E2 25271.657} C_VEL
LIN {X 0,Y 211.259,Z 1201.182,A -85,B 0,C 180,E1 25287.949,E2 25287.949} C_VEL
LIN {X 0,Y 210.728,Z 1202.231,A -85,B 0,C 180,E1 25303.475,E2 25303.475} C_VEL
LIN {X 0,Y 217.865,Z 1194.35,A -85,B 0,C 180,E1 25321.476,E2 25321.476} C_VEL
LIN {X 0,Y 244.297,Z 1171.945,A -85,B 0,C 180,E1 25340.898,E2 25340.898} C_VEL
LIN {X 0,Y 286.392,Z 1136.264,A -85,B 0,C 180,E1 25355.028,E2 25355.028} C_VEL
LIN {X 0,Y 335.603,Z 1087.175,A -85,B 0,C 180,E1 25364.536,E2 25364.536} C_VEL
LIN {X 0,Y 381.245,Z 1029.159,A -85,B 0,C 180,E1 25370.364,E2 25370.364} C_VEL
LIN {X 0,Y 384.941,Z 1022.982,A -85,B 0,C 180,E1 25371.094,E2 25371.094} C_VEL
LIN {X 0,Y 386.396,Z 1011.329,A -85,B 0,C 180,E1 25378.853,E2 25378.853} C_VEL
LIN {X 0,Y 386.41,Z 1010.943,A -85,B 0,C 180,E1 25385.609,E2 25385.609} C_VEL
LIN {X 0,Y 385.743,Z 1022.445,A -85,B 0,C 180,E1 25394.181,E2 25394.181} C_VEL
LIN {X 0,Y 383.643,Z 1026.823,A -85,B 0,C 180,E1 25395.04,E2 25395.04} C_VEL
LIN {X 0,Y 337.857,Z 1086.38,A -85,B 0,C 180,E1 25400.734,E2 25400.734} C_VEL
LIN {X 0,Y 288.026,Z 1137.069,A -85,B 0,C 180,E1 25410.086,E2 25410.086} C_VEL
LIN {X 0,Y 244.401,Z 1174.851,A -85,B 0,C 180,E1 25424.468,E2 25424.468} C_VEL
LIN {X 0,Y 218.366,Z 1197.596,A -85,B 0,C 180,E1 25443.16,E2 25443.16} C_VEL
LIN {X 0,Y 211.324,Z 1206.062,A -85,B 0,C 180,E1 25459.659,E2 25459.659} C_VEL
LIN {X 0,Y 210.973,Z 1206.998,A -85,B 0,C 180,E1 25472.054,E2 25472.054} C_VEL
LIN {X 0,Y 213.573,Z 1200.823,A -85,B 0,C 180,E1 25488.628,E2 25488.628} C_VEL
LIN {X 0,Y 230.118,Z 1181.31,A -85,B 0,C 180,E1 25507.992,E2 25507.992} C_VEL
LIN {X 0,Y 264.504,Z 1147.25,A -85,B 0,C 180,E1 25524.07,E2 25524.07} C_VEL
LIN {X 0,Y 308.999,Z 1099.568,A -85,B 0,C 180,E1 25535.209,E2 25535.209} C_VEL
LIN {X 0,Y 353.802,Z 1040.042,A -85,B 0,C 180,E1 25542.488,E2 25542.488} C_VEL
LIN {X 0,Y 371.654,Z 1010.135,A -85,B 0,C 180,E1 25545.054,E2 25545.054} C_VEL
LIN {X 0,Y 371.475,Z 990.887,A -85,B 0,C 180,E1 25552.987,E2 25552.987} C_VEL
LIN {X 0,Y 371.591,Z 981.218,A -85,B 0,C 180,E1 25561.193,E2 25561.193} C_VEL
LIN {X 0,Y 370.734,Z 985.72,A -85,B 0,C 180,E1 25569.443,E2 25569.443} C_VEL
LIN {X 0,Y 370.746,Z 1001.191,A -85,B 0,C 180,E1 25577.894,E2 25577.894} C_VEL
LIN {X 0,Y 369.264,Z 1013.553,A -85,B 0,C 180,E1 25581.762,E2 25581.762} C_VEL
LIN {X 0,Y 326.977,Z 1075.486,A -85,B 0,C 180,E1 25587.85,E2 25587.85} C_VEL
LIN {X 0,Y 321.621,Z 1082.107,A -85,B 0,C 180,E1 25588.76,E2 25588.76} C_VEL
LIN {X 0,Y 298.131,Z 1105.384,A -85,B 0,C 180,E1 25591.158,E2 25591.158} C_VEL
LIN {X 0,Y 254.058,Z 1149.733,A -85,B 0,C 180,E1 25602.788,E2 25602.788} C_VEL
LIN {X 0,Y 219.652,Z 1181.688,A -85,B 0,C 180,E1 25620.143,E2 25620.143} C_VEL
LIN {X 0,Y 205.045,Z 1197.91,A -85,B 0,C 180,E1 25639.351,E2 25639.351} C_VEL
LIN {X 0,Y 202.987,Z 1202.318,A -85,B 0,C 180,E1 25652.147,E2 25652.147} C_VEL
LIN {X 0,Y 203.878,Z 1200.987,A -85,B 0,C 180,E1 25669.562,E2 25669.562} C_VEL
LIN {X 0,Y 218.329,Z 1187.881,A -85,B 0,C 180,E1 25690.391,E2 25690.391} C_VEL
LIN {X 0,Y 254.57,Z 1159.498,A -85,B 0,C 180,E1 25708.717,E2 25708.717} C_VEL
LIN {X 0,Y 303.794,Z 1117.094,A -85,B 0,C 180,E1 25721.032,E2 25721.032} C_VEL
LIN {X 0,Y 354.278,Z 1062.838,A -85,B 0,C 180,E1 25728.75,E2 25728.75} C_VEL
LIN {X 0,Y 380.221,Z 1027.703,A -85,B 0,C 180,E1 25731.951,E2 25731.951} C_VEL
LIN {X 0,Y 381.788,Z 1017.964,A -85,B 0,C 180,E1 25738.839,E2 25738.839} C_VEL
LIN {X 0,Y 381.853,Z 1017.62,A -85,B 0,C 180,E1 25745.676,E2 25745.676} C_VEL
LIN {X 0,Y 380.799,Z 1028.236,A -85,B 0,C 180,E1 25753.803,E2 25753.803} C_VEL
LIN {X 0,Y 332.419,Z 1089.568,A -85,B 0,C 180,E1 25759.788,E2 25759.788} C_VEL
LIN {X 0,Y 281.821,Z 1139.13,A -85,B 0,C 180,E1 25769.123,E2 25769.123} C_VEL
LIN {X 0,Y 236.352,Z 1176.771,A -85,B 0,C 180,E1 25784.074,E2 25784.074} C_VEL
LIN {X 0,Y 209.742,Z 1198.823,A -85,B 0,C 180,E1 25803.798,E2 25803.798} C_VEL
LIN {X 0,Y 203.046,Z 1206.848,A -85,B 0,C 180,E1 25823.562,E2 25823.562} C_VEL
LIN {X 0,Y 203.038,Z 1206.128,A -85,B 0,C 180,E1 25836.426,E2 25836.426} C_VEL
LIN {X 0,Y 208.478,Z 1196.959,A -85,B 0,C 180,E1 25854.666,E2 25854.666} C_VEL
LIN {X 0,Y 232.278,Z 1172.899,A -85,B 0,C 180,E1 25874.412,E2 25874.412} C_VEL
LIN {X 0,Y 273.032,Z 1133.916,A -85,B 0,C 180,E1 25889.408,E2 25889.408} C_VEL
LIN {X 0,Y 320.011,Z 1081.999,A -85,B 0,C 180,E1 25899.205,E2 25899.205} C_VEL
LIN {X 0,Y 363.509,Z 1020.718,A -85,B 0,C 180,E1 25905.241,E2 25905.241} C_VEL
LIN {X 0,Y 366.738,Z 1015.268,A -85,B 0,C 180,E1 25905.657,E2 25905.657} C_VEL
LIN {X 0,Y 367.057,Z 996.01,A -85,B 0,C 180,E1 25914.094,E2 25914.094} C_VEL
LIN {X 0,Y 367.443,Z 988.116,A -85,B 0,C 180,E1 25921.206,E2 25921.206} C_VEL
LIN {X 0,Y 366.466,Z 992.736,A -85,B 0,C 180,E1 25929.554,E2 25929.554} C_VEL
LIN {X 0,Y 365.874,Z 1008.711,A -85,B 0,C 180,E1 25938.141,E2 25938.141} C_VEL
LIN {X 0,Y 364.904,Z 1016.74,A -85,B 0,C 180,E1 25940.774,E2 25940.774} C_VEL
LIN {X 0,Y 321.741,Z 1077.941,A -85,B 0,C 180,E1 25946.831,E2 25946.831} C_VEL
LIN {X 0,Y 298.131,Z 1105.384,A -85,B 0,C 180,E1 25951.158,E2 25951.158} C_VEL
LIN {X 0,Y 273.766,Z 1126.413,A -85,B 0,C 180,E1 25954.172,E2 25954.172} C_VEL
LIN {X 0,Y 229.935,Z 1166.551,A -85,B 0,C 180,E1 25968.744,E2 25968.744} C_VEL
LIN {X 0,Y 203.023,Z 1191.024,A -85,B 0,C 180,E1 25988.077,E2 25988.077} C_VEL
LIN {X 0,Y 195.273,Z 1201.421,A -85,B 0,C 180,E1 26007.781,E2 26007.781} C_VEL
LIN {X 0,Y 194.517,Z 1202.554,A -85,B 0,C 180,E1 26022.699,E2 26022.699} C_VEL
LIN {X 0,Y 201.791,Z 1195.861,A -85,B 0,C 180,E1 26041.746,E2 26041.746} C_VEL
LIN {X 0,Y 229.681,Z 1174.766,A -85,B 0,C 180,E1 26062.409,E2 26062.409} C_VEL
LIN {X 0,Y 274.768,Z 1139.887,A -85,B 0,C 180,E1 26077.156,E2 26077.156} C_VEL
LIN {X 0,Y 326.82,Z 1091.523,A -85,B 0,C 180,E1 26086.737,E2 26086.737} C_VEL
LIN {X 0,Y 374.773,Z 1033.874,A -85,B 0,C 180,E1 26092.484,E2 26092.484} C_VEL
LIN {X 0,Y 376.953,Z 1024.422,A -85,B 0,C 180,E1 26098.824,E2 26098.824} C_VEL
LIN {X 0,Y 377.027,Z 1024.097,A -85,B 0,C 180,E1 26105.749,E2 26105.749} C_VEL
LIN {X 0,Y 375.976,Z 1033.158,A -85,B 0,C 180,E1 26112.97,E2 26112.97} C_VEL
LIN {X 0,Y 326.168,Z 1093.734,A -85,B 0,C 180,E1 26118.952,E2 26118.952} C_VEL
LIN {X 0,Y 273.976,Z 1142.623,A -85,B 0,C 180,E1 26128.52,E2 26128.52} C_VEL
LIN {X 0,Y 229.156,Z 1177.938,A -85,B 0,C 180,E1 26143.248,E2 26143.248} C_VEL
LIN {X 0,Y 201.355,Z 1199.758,A -85,B 0,C 180,E1 26164.139,E2 26164.139} C_VEL
LIN {X 0,Y 195.034,Z 1206.767,A -85,B 0,C 180,E1 26183.296,E2 26183.296} C_VEL
LIN {X 0,Y 195.028,Z 1206.016,A -85,B 0,C 180,E1 26196.691,E2 26196.691} C_VEL
LIN {X 0,Y 200.328,Z 1197.558,A -85,B 0,C 180,E1 26214.597,E2 26214.597} C_VEL
LIN {X 0,Y 224.053,Z 1174.646,A -85,B 0,C 180,E1 26234.75,E2 26234.75} C_VEL
LIN {X 0,Y 266.23,Z 1136.036,A -85,B 0,C 180,E1 26250.292,E2 26250.292} C_VEL
LIN {X 0,Y 314.304,Z 1084.828,A -85,B 0,C 180,E1 26260.181,E2 26260.181} C_VEL
